	DOH_Y56:=FALSE;
	Y73:=FALSE;	
	//不同蓄能器压力下马大排量电流和主泵供能系数AcPre_w的设置
	IF	GVL_SaveEngine.AI_PAcPre>280 THEN //全部改小0.05
		GVL_SaveEngine.PWM_Y33_SET_Target:=400;//排量120  396-378
		AcPre_w:=0.3;//0.35-0.3 
	ELSIF GVL_SaveEngine.AI_PAcPre>270 THEN
		GVL_SaveEngine.PWM_Y33_SET_Target:=375;//排量130  378-360
		AcPre_w:=0.3;//0.35-0.3//0.15-0.35-0.5-0.4-0.35
	ELSIF GVL_SaveEngine.AI_PAcPre>250 THEN
		GVL_SaveEngine.PWM_Y33_SET_Target:=350;//排量150  340-322 
		AcPre_w:=0.4;//0.4-0.3       //0.25-0.45-0.6-0.5-0.45
	ELSIF  GVL_SaveEngine.AI_PAcPre>230 THEN
		GVL_SaveEngine.PWM_Y33_SET_Target:=325;//排量165 313-295
		AcPre_w:=0.55;//0.5-0.4       //0.4-0.6-0.75-0.65-0.6
	ELSIF  GVL_SaveEngine.AI_PAcPre>220 THEN                               //新增
		GVL_SaveEngine.PWM_Y33_SET_Target:=275;//排量165   
		AcPre_w:=0.6;//0.5-0.4       //0.65
	ELSIF  GVL_SaveEngine.AI_PAcPre>210 THEN
		GVL_SaveEngine.PWM_Y33_SET_Target:=250;//排量190  287-269          //变269-248
		AcPre_w:=0.65;//         //0.55-0.75-0.9-0.8-0.75
	ELSIF GVL_SaveEngine.AI_PAcPre>205 THEN   //200-205 0426
		GVL_SaveEngine.PWM_Y33_SET_Target:=200;//排量200  249-230-248      //248-230
		AcPre_w:=0.7;//         0.6-0.8-0.95-0.85-0.8
	ELSIF GVL_SaveEngine.AI_PAcPre>200 THEN   //190-200 0426
		GVL_SaveEngine.PWM_Y33_SET_Target:=150;//排量210                //230-212
		AcPre_w:=0.75;          //0.7-0.9-1-0.95-0.9
	ELSIF  GVL_SaveEngine.AI_PAcPre>195 THEN  //180-195
		GVL_SaveEngine.PWM_Y33_SET_Target:=100;//排量216                 //230-200
		AcPre_w:=0.85;         //0.85-1
	ELSIF  GVL_SaveEngine.AI_PAcPre>190 THEN  //170-180
		GVL_SaveEngine.PWM_Y33_SET_Target:=100;//排量200
		AcPre_w:=0.9;//0.9-0.8
	ELSIF  GVL_SaveEngine.AI_PAcPre>180 THEN  //160-170
		GVL_SaveEngine.PWM_Y33_SET_Target:=100;//排量200
		AcPre_w:=1;
	ELSE
		GVL_SaveEngine.PWM_Y33_SET_Target:=100;//排量200
		AcPre_w:=1;
	END_IF


	//不同发动机转速下根据马达排量和目标转速计算出的主泵最大电流
  	CASE SPEED_CASE OF
	//                                    权重 速度v 转速n            主卷排量 v_winch
	1: CasePWM_Y1:=REAL_TO_UINT(362.5+47.8*AcPre_w*30/1100*(600-PWM_Y33_SET_Target)/1.85) ;//362.5+1350/转速*AcPre_w*排量
	2: CasePWM_Y1:=REAL_TO_UINT(362.5+47.8*AcPre_w*38/1200*(600-PWM_Y33_SET_Target)/1.85) ;//362.5+1710/转速*AcPre_w*排量
	3: CasePWM_Y1:=REAL_TO_UINT(362.5+47.8*AcPre_w*50/1450*(600-PWM_Y33_SET_Target)/1.85) ;//362.5+2250/转速*AcPre_w*排量
	4: CasePWM_Y1:=REAL_TO_UINT(362.5+47.8*AcPre_w*55/1600*(600-PWM_Y33_SET_Target)/1.85) ;//362.5+2475/转速*AcPre_w*排量
	5: CasePWM_Y1:=REAL_TO_UINT(362.5+47.8*AcPre_w*62/1800*(600-PWM_Y33_SET_Target)/1.85) ;//362.5+2790/转速*AcPre_w*排量
	6: CasePWM_Y1:=REAL_TO_UINT(362.5+47.8*AcPre_w*65/1900*(600-PWM_Y33_SET_Target)/1.85) ;//362.5+2925/转速*AcPre_w*排量
	END_CASE


CasePWM_Y1:=LIMIT(400,CasePWM_Y1,700);
PWM_Y1_Target:=REAL_TO_UINT(UINT_TO_REAL(CasePWM_Y1-PAR_Y1_NegFull)*PWM_JOYY_L_DOWN/1000+PAR_Y1_NegFull);
PWM_Y2_Target:=REAL_TO_UINT(UINT_TO_REAL(CasePWM_Y1-PAR_Y2_NegFull)*PWM_JOYY_L_DOWN/1000+PAR_Y2_NegFull);						

//主阀控制
PWM_Y7_SET_Target:=REAL_TO_UINT(UINT_TO_REAL(PWM_JOYY_L_DOWN)/1000*(PAR_Valve1_PosFull-PAR_Valve2_NegFull)+PAR_Valve2_NegFull);
PWM_Y9_SET_Target:=REAL_TO_UINT(UINT_TO_REAL(PWM_JOYY_L_DOWN)/1000*(PAR_Valve2_PosFull-PAR_Valve2_NegFull)+PAR_Valve2_NegFull);
PWM_Y8_SET:=0;
PWM_Y10_SET:=0;
	
IF PWM_Y33_SET>=PWM_Y33_SET_Target THEN
	PWM_Y33_SET := PWM_Y33_SET_Target;
END_IF
	
IF(PWM_Y33_SET<PWM_Y33_SET_Target) THEN
	PWM_Y33_SET:=REAL_TO_UINT(UINT_TO_REAL(PWM_Y33_SET)+JianGE6);
END_IF

IF DIL_SQ3 THEN
	PWM_Y33_SET:=0;
END_IF
(*主泵功率控制,屏蔽了Pressure_Coe,2模式没有进行恒功率控制，仅保留斜坡*)

//区分发动机转速
MainPump_Pressure_Taget1450:=PAR_NegFull_x;
MainPump_Pressure_Taget1600:=PAR_PosFull_x;
MainPump_Pressure_Taget1750:=PAR_Zero_x;
IF EngineSpeedTarget<=1080 THEN SPEED_CASE:=1;
ELSIF EngineSpeedTarget>1080 AND EngineSpeedTarget<=1300 THEN SPEED_CASE:=2;
ELSIF EngineSpeedTarget>1300 AND EngineSpeedTarget<=1520 THEN SPEED_CASE:=3;
ELSIF EngineSpeedTarget>1520 AND EngineSpeedTarget<=1680 THEN SPEED_CASE:=4;
ELSIF EngineSpeedTarget>1680 AND EngineSpeedTarget<=1820 THEN SPEED_CASE:=5;
ELSIF EngineSpeedTarget>1820 THEN SPEED_CASE:=6;;END_IF
//不同转速下的发动机最大功率*)
CASE SPEED_CASE OF
1:  Enginer_Power:=135;
2:  Enginer_Power:=174;
3:  Enginer_Power:=200;
4:  Enginer_Power:=230;
5:  Enginer_Power:=250;
6:  Enginer_Power:=261;
END_CASE
//不同转速下的压力值
IF(CANO_Fubeng_Press>100)THEN
	CASE SPEED_CASE OF
	1:MainPump_Pressure_Taget:=MainPump_Pressure_Taget1000-HELIU_Press_Target1000;
	2:MainPump_Pressure_Taget:=MainPump_Pressure_Taget1200-HELIU_Press_Target1200;
	3:MainPump_Pressure_Taget:=MainPump_Pressure_Taget1450-HELIU_Press_Target1400;
	4:MainPump_Pressure_Taget:=MainPump_Pressure_Taget1600-HELIU_Press_Target1600;
	5:MainPump_Pressure_Taget:=MainPump_Pressure_Taget1750-HELIU_Press_Target1800;
	6:MainPump_Pressure_Taget:=MainPump_Pressure_Taget1900-HELIU_Press_Target1900;
	END_CASE
ELSE
	CASE SPEED_CASE OF
	1:MainPump_Pressure_Taget:=MainPump_Pressure_Taget1000;
	2:MainPump_Pressure_Taget:=MainPump_Pressure_Taget1200;
	3:MainPump_Pressure_Taget:=MainPump_Pressure_Taget1450;
	4:MainPump_Pressure_Taget:=MainPump_Pressure_Taget1600;
	5:MainPump_Pressure_Taget:=MainPump_Pressure_Taget1750;
	6:MainPump_Pressure_Taget:=MainPump_Pressure_Taget1900;
	END_CASE		
END_IF

IF( CANI_ECOSwitch) THEN
	CASE SPEED_CASE OF
	1:MainPump_Pressure_Taget:=MainPump_Pressure_Taget1000-ECO_Press_Target1000;
	2:MainPump_Pressure_Taget:=MainPump_Pressure_Taget1200-ECO_Press_Target1200;
	3:MainPump_Pressure_Taget:=MainPump_Pressure_Taget1450-ECO_Press_Target1400;
	4:MainPump_Pressure_Taget:=MainPump_Pressure_Taget1600-ECO_Press_Target1600;
	5:MainPump_Pressure_Taget:=MainPump_Pressure_Taget1750-ECO_Press_Target1800;
	6:MainPump_Pressure_Taget:=MainPump_Pressure_Taget1900-ECO_Press_Target1900;
	END_CASE
END_IF
MainPump_Pressure:=CANO_MainPUMP_Press1+CANO_MainPUMP_Press2;
//消除滤波
MainPump_Pressure_Subtract:= UINT_TO_INT(MainPump_Pressure-MainPump_Pressure_last1);


//大范围波动
IF MainPump_Pressure_Subtract>270 OR MainPump_Pressure_Subtract<-270 THEN
	Subtract:=TRUE;
ELSE
	Subtract:=FALSE;	
END_IF
	TIME_LvBo4(IN:=Subtract,PT:=T#10MS);
	
IF(TIME_LvBo4.Q) AND (CANO_MainPUMP_Press1>210) THEN 
		MainPump_Pressure_ChangeBool1:=TRUE;
END_IF
	TIME_LvBo1(IN:=MainPump_Pressure_ChangeBool1,PT:=T#2S);
IF(TIME_LvBo1.Q) THEN
	MainPump_Pressure_ChangeBool1 :=FALSE;
END_IF

IF(MainPump_Pressure_ChangeBool1) AND (MainPump_Pressure>MainPump_Pressure_last1) THEN 
	MainPump_Pressure_last1:=MainPump_Pressure;
END_IF

//小范围波动
t_powertime:=TO_TIME(PAR_DeadBand_x);
IF (NOT MainPump_Pressure_ChangeBool1) THEN
	IF(MainPump_Pressure_Subtract>40 OR MainPump_Pressure_Subtract<-40)THEN 
		MainPump_Pressure_ChangeBool:=TRUE;
	ELSE
		MainPump_Pressure_ChangeBool:=FALSE;
	END_IF

	TIME_LvBo2(IN:=MainPump_Pressure_ChangeBool,PT:=t_powertime);
	IF(TIME_LvBo2.Q )THEN
		MainPump_Pressure_last1:=MainPump_Pressure;
	END_IF	
END_IF


IF PowerHead_move AND NOT(MainWinch_move) THEN
		JianGE2:=0.005;
ELSE
	IF(EngineSpeedTarget>1000 AND EngineSpeedTarget<1300)THEN
		JianGE2:=0.005;
	ELSE
		JianGE2:=0.005;
	END_IF
END_IF
(*	
IF MainPump_Pressure_last1>MainPump_Pressure_Taget THEN
	Pressure_Coe_Taget:=UINT_TO_REAL(MainPump_Pressure_Taget)/UINT_TO_REAL(MainPump_Pressure_last1);(*压力系数*)
ELSE
	Pressure_Coe_Taget:=1;
END_IF
Pressure_Coe := Pressure_Coe_Taget;
*)

(*
Pressure_Coe := 1;
IF MainPump_Pressure_last1>MainPump_Pressure_Taget  THEN
	IF(PWM_Y1_Target>=PAR_Y1_1_NegFull)THEN
		PWM_Y1_Target_OutPut:=REAL_TO_UINT(UINT_TO_REAL(PWM_Y1_Target-PAR_Y1_1_NegFull)*Pressure_Coe+PAR_Y1_1_NegFull);
	END_IF
	IF(PWM_Y2_Target>=PAR_Y1_1_NegFull)THEN
		PWM_Y2_Target_OutPut:=REAL_TO_UINT(UINT_TO_REAL(PWM_Y2_Target-PAR_Y1_1_NegFull)*Pressure_Coe+PAR_Y1_1_NegFull);
	END_IF
ELSE
	PWM_Y1_Target_OutPut:=PWM_Y1_Target;
	PWM_Y2_Target_OutPut:=PWM_Y2_Target;
END_IF
*)

PWM_Y1_Target_OutPut:=PWM_Y1_Target;
PWM_Y2_Target_OutPut:=PWM_Y2_Target;
IF(EngineSpeedTarget>CANO_SPEED AND CANO_SPEED>400)THEN
	EngineSpeedSub:=EngineSpeedTarget - CANO_SPEED;
ELSE
	EngineSpeedSub:=0;
END_IF

IF(PWM_Y1_Target_OutPut<300)THEN PWM_Y1_Target_OutPut:=300;END_IF	
IF(PWM_Y2_Target_OutPut<300)THEN PWM_Y2_Target_OutPut:=300;END_IF

RAMP15_IN:=PWM_Y1_Target_OutPut;
RAMP16_IN:=PWM_Y2_Target_OutPut;
(*
IF MainWinch_move  OR  LeftMove_move OR RightMove_move THEN  
	TIMEBASE_pump:=T#1000MS;
	TIMEBASE_xiehe:=T#500MS;
ELSE
	TIMEBASE_pump:=T#400MS;
	TIMEBASE_xiehe:=T#200MS;
END_IF
t_PowerHead_move(IN:= MainWinch_move,PT:=T#2S);
IF t_PowerHead_move.Q THEN
	F_RAMP_pump:=x_t_PowerHead_move;
	R_RAMP_pump:=x2_t_PowerHead_move;
ELSE
	F_RAMP_pump:=1000;
	R_RAMP_pump:=300;
END_IF
*)
(*
//减斜坡800->2000
RAMP15(
	IN:=UINT_TO_INT(RAMP15_IN), 
	ASCEND:= 300, 
	DESCEND:= 2000, 
	TIMEBASE:=T#1000MS , 
	RESET:=FALSE , 
	OUT=>(PWM_Y1_SET));
	
RAMP16(
	IN:=UINT_TO_INT(RAMP16_IN), 
	ASCEND:= 300, 
	DESCEND:= 2000, 
	TIMEBASE:=T#1000MS , 
	RESET:=FALSE , 
	OUT=>(PWM_Y2_SET));
*)
	CASE SPEED_CASE OF
                1:F_RAMP_pump:=1500; R_RAMP_pump:=100;                  
                2: 		IF MainWinch_move AND (JiaYa_move OR CANO_JiayaPressure>80)  THEN    //3泵同时起压时，降低主泵的加载速度，避免掉速熄火
                                F_RAMP_pump:=1500; R_RAMP_pump:=100;
                        ELSE
                                F_RAMP_pump:=1500; R_RAMP_pump:=100;//从200降
                                IF  PWM_JOYY_L_UP>10 THEN
                                 F_RAMP_pump:=1500; R_RAMP_pump:=200;
                                END_IF
                        END_IF            
                3:
                        IF MainWinch_move AND (JiaYa_move OR CANO_JiayaPressure>80)  THEN    //3泵同时起压时，降低主泵的加载速度，避免掉速熄火
                                F_RAMP_pump:=1500; R_RAMP_pump:=150;
                        ELSE
                                F_RAMP_pump:=1500; R_RAMP_pump:=TO_INT(PAR_NegFull_y);
                                IF  PWM_JOYY_L_UP>10 THEN
                                 F_RAMP_pump:=1500; R_RAMP_pump:=300;
                                END_IF
                        END_IF                
                4:
                        IF MainWinch_move AND (JiaYa_move OR CANO_JiayaPressure>80)  THEN
                                F_RAMP_pump:=1500; R_RAMP_pump:=150;
                        ELSE
                                F_RAMP_pump:=1500; R_RAMP_pump:=TO_INT(PAR_PosFull_y);//从200降
                                IF  PWM_JOYY_L_UP>10 THEN
                                 F_RAMP_pump:=1500; R_RAMP_pump:=300;
                                END_IF
                        END_IF                                
                5:
                        IF MainWinch_move AND (JiaYa_move OR CANO_JiayaPressure>80)  THEN
                                F_RAMP_pump:=1500; R_RAMP_pump:=200;
                        ELSE
                                F_RAMP_pump:=1500; R_RAMP_pump:=TO_INT(PAR_Zero_y);
                                IF  PWM_JOYY_L_UP>10 THEN
                                 F_RAMP_pump:=1500; R_RAMP_pump:=300;
                                END_IF
                        END_IF                        
                6:		IF MainWinch_move AND (JiaYa_move OR CANO_JiayaPressure>80)  THEN
                                F_RAMP_pump:=1500; R_RAMP_pump:=200;
                        ELSE
                                F_RAMP_pump:=1500; R_RAMP_pump:=200;
                                IF  PWM_JOYY_L_UP>10 THEN
                                 F_RAMP_pump:=1500; R_RAMP_pump:=300;
                                END_IF
                        END_IF	
	END_CASE
(******斜坡增步长300 斜坡降步长300->400*****)	
RAMP15(
	IN:=UINT_TO_INT(RAMP15_IN), 
	ASCEND:= R_RAMP_pump, 
	DESCEND:= 2000, //3切2模式时 速度变快 降低主泵电流变化速度 
	TIMEBASE:=T#1000MS , 
	RESET:=FALSE , 
	OUT=>(PWM_Y1_SET));
(******减斜坡300->400*****)	
RAMP16(
	IN:=UINT_TO_INT(RAMP16_IN), 
	ASCEND:= R_RAMP_pump, 
	DESCEND:= 2000, 
	TIMEBASE:=T#1000MS , 
	RESET:=FALSE , 
	OUT=>(PWM_Y2_SET));


IF (NOT Rotation_move) AND (NOT MainWinch_move) AND (NOT PowerHead_move)
		AND (NOT JiaYa_move) AND (NOT ViceWinch_move)
		AND (NOT LeftMove_move) AND (NOT RightMove_move)  THEN
	PWM_Y1_Target:=0;
	PWM_Y2_Target:=0;
END_IF


IF PWM_Y1_SET<TO_INT(PAR_Y1_1_NegFull )THEN
	PWM_Y1_SET:=TO_INT(PAR_Y1_1_NegFull);
END_IF

IF PWM_Y2_SET<TO_INT(PAR_Y1_1_NegFull )THEN
	PWM_Y2_SET:=TO_INT(PAR_Y1_1_NegFull);
END_IF

IF(PWM_Y1_SET>1000) THEN
	PWM_Y1_SET := 300;
END_IF

IF(PWM_Y2_SET>1000) THEN
	PWM_Y2_SET := 300;
END_IF	
  //Y7 8 9 10处理	
		IF(PWM_Y8_SET<1000  AND  PWM_Y8_SET>=900)THEN    //主卷下放斜坡值
				F_RAMP_mainwinch_down:=200;
			
			ELSIF(PWM_Y8_SET<900)THEN
				F_RAMP_mainwinch_down:=400;
			ELSE
				F_RAMP_mainwinch_down:=400;
			END_IF
			
		IF(PWM_Y7_SET<1000  AND  PWM_Y7_SET>=900)THEN  //主卷上提斜坡值
				F_RAMP_mainwinch_down:=300;
		ELSIF(PWM_Y7_SET<900  )THEN
				F_RAMP_mainwinch_down:=200;
		ELSE
				F_RAMP_mainwinch_down:=400;
		END_IF
			
	RAMP7(
		IN:=WORD_TO_INT(PWM_Y7_SET_Target), 
		ASCEND:= R_RAMP_mainwinch, 
		DESCEND:= F_RAMP_mainwinch_up, 
		TIMEBASE:=TIMEBASE_mainwinch , 
		RESET:=FALSE , 
		OUT=>(PWM_Y7_SET_Target1));
	IF(PWM_Y7_SET_Target1>=400) THEN
		Curve_input:=TO_UINT(PWM_Y7_SET_Target1 - 400);
		IF(Curve_input>900) THEN
			Curve_input:=900;
		END_IF
		curve7(input:=REAL_TO_UINT(UINT_TO_REAL(Curve_input)*72.8),Zero:=FALSE,Full:=FALSE,
			   PAR_Progression:=Curve_Par,OutputEnable:=TRUE);
		PWM_Y7_SET:=PAR_Valve1_NegFull + REAL_TO_UINT(UINT_TO_REAL(curve7.Output)/72.8);
	ELSE
		PWM_Y7_SET:=0;
	END_IF
	
(*	
	RAMP8(
		IN:=WORD_TO_INT(PWM_Y8_SET_Target), 
		ASCEND:= R_RAMP_mainwinch, 
		DESCEND:= F_RAMP_mainwinch_down, 
		TIMEBASE:=TIMEBASE_mainwinch , 
		RESET:=FALSE , 
		OUT=>(PWM_Y8_SET_Target1));
	IF(PWM_Y8_SET_Target1>=400) THEN
		Curve_input:=TO_UINT(PWM_Y8_SET_Target1 - 400);
		IF(Curve_input>900) THEN
			Curve_input:=900;
		END_IF
		curve8(input:=REAL_TO_UINT(UINT_TO_REAL(Curve_input)*72.8),Zero:=FALSE,Full:=FALSE,
			   PAR_Progression:=Curve_Par,OutputEnable:=TRUE);
		PWM_Y8_SET:=PAR_Valve1_NegFull + REAL_TO_UINT(UINT_TO_REAL(curve8.Output)/72.8);
	ELSE
		PWM_Y8_SET:=0;
	END_IF
*)	
	
	RAMP9(
		IN:=WORD_TO_INT(PWM_Y9_SET_Target), 
		ASCEND:= R_RAMP_mainwinch, 
		DESCEND:= F_RAMP_mainwinch_up, 
		TIMEBASE:=TIMEBASE_mainwinch , 
		RESET:=FALSE , 
		OUT=>(PWM_Y9_SET_Target1));
	IF(PWM_Y9_SET_Target1>=400) THEN
		Curve_input:=TO_UINT(PWM_Y9_SET_Target1 - 400);
		IF(Curve_input>900) THEN
			Curve_input:=900;
		END_IF
		curve9(input:=REAL_TO_UINT(UINT_TO_REAL(Curve_input)*72.8),Zero:=FALSE,Full:=FALSE,
			   PAR_Progression:=Curve_Par,OutputEnable:=TRUE);
		PWM_Y9_SET:=PAR_Valve1_NegFull + REAL_TO_UINT(UINT_TO_REAL(curve9.Output)/72.8);
	ELSE
		PWM_Y9_SET:=0;
	END_IF
(*	
	RAMP10(
		IN:=WORD_TO_INT(PWM_Y10_SET_Target), 
		ASCEND:= R_RAMP_mainwinch, 
		DESCEND:= F_RAMP_mainwinch_down, 
		TIMEBASE:=TIMEBASE_mainwinch , 
		RESET:=FALSE , 
		OUT=>(PWM_Y10_SET_Target1));
	IF(PWM_Y10_SET_Target1>=400) THEN
		Curve_input:=TO_UINT(PWM_Y10_SET_Target1 - 400);
		IF(Curve_input>900) THEN
			Curve_input:=900;
		END_IF
		curve10(input:=REAL_TO_UINT(UINT_TO_REAL(Curve_input)*72.8),Zero:=FALSE,Full:=FALSE,
			   PAR_Progression:=Curve_Par,OutputEnable:=TRUE);
		PWM_Y10_SET:=PAR_Valve1_NegFull + REAL_TO_UINT(UINT_TO_REAL(curve10.Output)/72.8);
	ELSE
		PWM_Y10_SET:=0;
	END_IF
*)
    //Y7 8 9 10范围限制
	IF(PWM_Y7_SET>1300)THEN
		PWM_Y7_SET :=1300;
	END_IF
	IF(PWM_Y8_SET>1300)THEN
		PWM_Y8_SET :=1300;
	END_IF
	IF(PWM_Y9_SET>1300)THEN
		PWM_Y9_SET :=1300;
	END_IF
	IF(PWM_Y10_SET>1300)THEN
		PWM_Y10_SET :=1300;
	END_IF
	
	IF(PWM_Y7_SET<=300)THEN
		PWM_Y7_SET :=0;
	END_IF
	IF(PWM_Y8_SET<=300)THEN
		PWM_Y8_SET :=0;
	END_IF
	IF(PWM_Y9_SET<=300)THEN
		PWM_Y9_SET :=0;
	END_IF
	IF(PWM_Y10_SET<=300)THEN
		PWM_Y10_SET :=0;
	END_IF
	(*主泵卸荷阀控制*)
		//PWM_Y39_SET_Target:=MAX(PWM_Y8_SET,PWM_Y7_SET_Target);//直接给输出卸荷
		PWM_Y40_SET_Target:=MAX(PWM_Y9_SET_Target,PWM_Y10_SET);
	//(*卸荷动作缓冲*)
(*RAMP19(
	IN:=WORD_TO_INT(PWM_Y39_SET_Target), 
	ASCEND:= R_RAMP_xiehe, 
	DESCEND:= F_RAMP_xiehe, 
	TIMEBASE:=TIMEBASE_xiehe , 
	RESET:=FALSE , 
	OUT=>(PWM_Y39_SET_Target1));
IF(PWM_Y39_SET_Target1>=400) THEN
	Curve_input:=TO_UINT(PWM_Y39_SET_Target1 - 400);
	IF(Curve_input>900) THEN
		Curve_input:=900;
	END_IF
	curve19(input:=REAL_TO_UINT(UINT_TO_REAL(Curve_input)*72.8),Zero:=FALSE,Full:=FALSE,
		   PAR_Progression:=Curve_Par1,OutputEnable:=TRUE);
	PWM_Y39_SET:=PAR_Valve1_NegFull + REAL_TO_UINT(UINT_TO_REAL(curve19.Output)/72.8);
ELSE
	PWM_Y39_SET:=0;
END_IF
*)

RAMP20(
	IN:=WORD_TO_INT(PWM_Y40_SET_Target), 
	ASCEND:= R_RAMP_xiehe, 
	DESCEND:= F_RAMP_xiehe, 
	TIMEBASE:=TIMEBASE_xiehe , 
	RESET:=FALSE , 
	OUT=>(PWM_Y40_SET_Target1));
IF(PWM_Y40_SET_Target1>=400) THEN
	Curve_input:=TO_UINT(PWM_Y40_SET_Target1 - 400);
	IF(Curve_input>900) THEN
		Curve_input:=900;
	END_IF
	curve20(input:=REAL_TO_UINT(UINT_TO_REAL(Curve_input)*72.8),Zero:=FALSE,Full:=FALSE,
		   PAR_Progression:=Curve_Par1,OutputEnable:=TRUE);
	PWM_Y40_SET:=PAR_Valve1_NegFull + REAL_TO_UINT(UINT_TO_REAL(curve20.Output)/72.8);
ELSE
	PWM_Y40_SET:=0;
END_IF

IF(PWM_Y39_SET>1300)THEN
	PWM_Y39_SET :=1300;
END_IF
IF(PWM_Y40_SET>1300)THEN
	PWM_Y40_SET :=1300;
END_IF

IF(PWM_Y39_SET<=300)THEN
	PWM_Y39_SET :=0;
END_IF
IF(PWM_Y40_SET<=300)THEN
	PWM_Y40_SET :=0;
END_IF

END_PROGRAM

// StandardPLC/Application/SaveEngine/SaveEngineMode_3
PROGRAM SaveEngineMode_3
VAR
	PressLvBo_TON:TON;
	PressLvBo_TON1: TON;
	PressLvBo_TON2: TON;
	PressLvBo_TON3: TON;

END_VAR


(*******************节能控制阀主阀主泵输出执行**************************)
	
//ELSIF(GVL_SaveEngine.SaveEngineMode=3)THEN//上升能量不足模式
	GVL_SaveEngine.Y72OutPutState:=0;
	GVL_SaveEngine.Y71OutPutState:=0;
	DOH_Y56:=FALSE;
		Y73:=FALSE;	
	PWM_Y1_Target:=REAL_TO_UINT(UINT_TO_REAL(PWM_JOYY_L_DOWN)/1000*0.9*(PAR_Y1_PosFull-PAR_Y1_NegFull)+PAR_Y1_NegFull);
	PWM_Y2_Target:=REAL_TO_UINT(UINT_TO_REAL(PWM_JOYY_L_DOWN)/1000*0.9*(PAR_Y2_PosFull-PAR_Y2_NegFull)+PAR_Y2_NegFull);
	PWM_Y7_SET_Target:=REAL_TO_UINT(UINT_TO_REAL(PWM_JOYY_L_DOWN)/1000*(PAR_Valve1_PosFull-PAR_Valve2_NegFull)+PAR_Valve2_NegFull);
	PWM_Y9_SET_Target:=REAL_TO_UINT(UINT_TO_REAL(PWM_JOYY_L_DOWN)/1000*(PAR_Valve2_PosFull-PAR_Valve2_NegFull)+PAR_Valve2_NegFull);
	PWM_Y8_SET_Target:=300;
	PWM_Y10_SET_Target:=300;		
	(*电控马达主卷变量控制*)
	
PressLvBo_TON(IN:=CANO_ZhuJuanPressure>310,PT:=T#300MS);
PressLvBo_TON1(IN:=CANO_ZhuJuanPressure>290 AND CANO_ZhuJuanPressure<=310,PT:=T#300MS);
PressLvBo_TON2(IN:=CANO_ZhuJuanPressure>270 AND CANO_ZhuJuanPressure<=290,PT:=T#300MS);
PressLvBo_TON3(IN:=CANO_ZhuJuanPressure>250 AND CANO_ZhuJuanPressure<=270,PT:=T#300MS);
IF(CANO_ZhuJuanPressure>310 AND PressLvBo_TON.Q) OR P31_Flag THEN
        PWM_Y33_SET_Target :=230;   //排量200
        P31_Flag:=TRUE;
        IF (CANO_ZhuJuanPressure<270) THEN
                P31_Flag:=FALSE;        
        END_IF
ELSIF(CANO_ZhuJuanPressure>290 AND PressLvBo_TON1.Q) OR P29_Flag THEN   
        PWM_Y33_SET_Target :=267;   //排量180
        P29_Flag:=TRUE; 
        IF (CANO_ZhuJuanPressure<250) THEN
                P29_Flag:=FALSE; 
        END_IF
ELSIF(CANO_ZhuJuanPressure>270 AND PressLvBo_TON2.Q) OR P27_Flag THEN   
        PWM_Y33_SET_Target :=304;  //排量160
        P27_Flag:=TRUE;
        IF (CANO_ZhuJuanPressure<230) THEN
                P27_Flag:=FALSE; 
        END_IF
ELSIF(CANO_ZhuJuanPressure>250 AND PressLvBo_TON3.Q) OR P25_Flag THEN //压力小于270   
        PWM_Y33_SET_Target :=340;  //排量140
        P25_Flag:=TRUE; 
        IF (CANO_ZhuJuanPressure<210) THEN
                P25_Flag:=FALSE; 
        END_IF
ELSE //(CANO_ZhuJuanPressure<=250) THEN
        PWM_Y33_SET_Target :=370;
END_IF
	(*IF BiaoZHI_MainWinchUp THEN
		PWM_Y33_SET_Target:=370;
	END_IF
	*)
	  //Y33输出处理
	IF PWM_Y33_SET>=PWM_Y33_SET_Target THEN
	PWM_Y33_SET := PWM_Y33_SET_Target;
	END_IF
		
	IF(PWM_Y33_SET<PWM_Y33_SET_Target) THEN
		PWM_Y33_SET:=REAL_TO_UINT(UINT_TO_REAL(PWM_Y33_SET)+JianGE6);
	END_IF
	
	IF DIL_SQ3 THEN
		PWM_Y33_SET:=0;
	END_IF
	
(*主泵功率控制*)

//区分发动机转速
MainPump_Pressure_Taget1450:=PAR_NegFull_x;
MainPump_Pressure_Taget1600:=PAR_PosFull_x;
MainPump_Pressure_Taget1750:=PAR_Zero_x;
IF EngineSpeedTarget<=1080 THEN SPEED_CASE:=1;
ELSIF EngineSpeedTarget>1080 AND EngineSpeedTarget<=1300 THEN SPEED_CASE:=2;
ELSIF EngineSpeedTarget>1300 AND EngineSpeedTarget<=1520 THEN SPEED_CASE:=3;
ELSIF EngineSpeedTarget>1520 AND EngineSpeedTarget<=1680 THEN SPEED_CASE:=4;
ELSIF EngineSpeedTarget>1680 AND EngineSpeedTarget<=1820 THEN SPEED_CASE:=5;
ELSIF EngineSpeedTarget>1820 THEN SPEED_CASE:=6;;END_IF
//不同转速下的发动机最大功率*)
CASE SPEED_CASE OF
1:  Enginer_Power:=135;
2:  Enginer_Power:=174;
3:  Enginer_Power:=200;
4:  Enginer_Power:=230;
5:  Enginer_Power:=250;
6:  Enginer_Power:=261;
END_CASE
//不同转速下的压力值
IF(CANO_Fubeng_Press>100)THEN
	CASE SPEED_CASE OF
	1:MainPump_Pressure_Taget:=MainPump_Pressure_Taget1000-HELIU_Press_Target1000;
	2:MainPump_Pressure_Taget:=MainPump_Pressure_Taget1200-HELIU_Press_Target1200;
	3:MainPump_Pressure_Taget:=MainPump_Pressure_Taget1450-HELIU_Press_Target1400;
	4:MainPump_Pressure_Taget:=MainPump_Pressure_Taget1600-HELIU_Press_Target1600;
	5:MainPump_Pressure_Taget:=MainPump_Pressure_Taget1750-HELIU_Press_Target1800;
	6:MainPump_Pressure_Taget:=MainPump_Pressure_Taget1900-HELIU_Press_Target1900;
	END_CASE
ELSE
	CASE SPEED_CASE OF
	1:MainPump_Pressure_Taget:=MainPump_Pressure_Taget1000;
	2:MainPump_Pressure_Taget:=MainPump_Pressure_Taget1200;
	3:MainPump_Pressure_Taget:=MainPump_Pressure_Taget1450;
	4:MainPump_Pressure_Taget:=MainPump_Pressure_Taget1600;
	5:MainPump_Pressure_Taget:=MainPump_Pressure_Taget1750;
	6:MainPump_Pressure_Taget:=MainPump_Pressure_Taget1900;
	END_CASE		
END_IF

IF( CANI_ECOSwitch) THEN
	CASE SPEED_CASE OF
	1:MainPump_Pressure_Taget:=MainPump_Pressure_Taget1000-ECO_Press_Target1000;
	2:MainPump_Pressure_Taget:=MainPump_Pressure_Taget1200-ECO_Press_Target1200;
	3:MainPump_Pressure_Taget:=MainPump_Pressure_Taget1450-ECO_Press_Target1400;
	4:MainPump_Pressure_Taget:=MainPump_Pressure_Taget1600-ECO_Press_Target1600;
	5:MainPump_Pressure_Taget:=MainPump_Pressure_Taget1750-ECO_Press_Target1800;
	6:MainPump_Pressure_Taget:=MainPump_Pressure_Taget1900-ECO_Press_Target1900;
	END_CASE
END_IF
MainPump_Pressure:=CANO_MainPUMP_Press1+CANO_MainPUMP_Press2;
//消除滤波
MainPump_Pressure_Subtract:= UINT_TO_INT(MainPump_Pressure-MainPump_Pressure_last1);


//大范围波动
IF MainPump_Pressure_Subtract>270 OR MainPump_Pressure_Subtract<-270 THEN
	Subtract:=TRUE;
ELSE
	Subtract:=FALSE;	
END_IF
	TIME_LvBo4(IN:=Subtract,PT:=T#10MS);
	
IF(TIME_LvBo4.Q) AND (CANO_MainPUMP_Press1>210) THEN 
	MainPump_Pressure_ChangeBool1:=TRUE;
END_IF
	TIME_LvBo1(IN:=MainPump_Pressure_ChangeBool1,PT:=T#2S);
IF(TIME_LvBo1.Q) THEN
	MainPump_Pressure_ChangeBool1 :=FALSE;
END_IF

IF(MainPump_Pressure_ChangeBool1) AND (MainPump_Pressure>MainPump_Pressure_last1) THEN 
	MainPump_Pressure_last1:=MainPump_Pressure;
END_IF

//小范围波动
t_powertime:=TO_TIME(PAR_DeadBand_x);
IF (NOT MainPump_Pressure_ChangeBool1) THEN
	IF(MainPump_Pressure_Subtract>40 OR MainPump_Pressure_Subtract<-40)THEN 
		MainPump_Pressure_ChangeBool:=TRUE;
	ELSE
		MainPump_Pressure_ChangeBool:=FALSE;
	END_IF

	TIME_LvBo2(IN:=MainPump_Pressure_ChangeBool,PT:=t_powertime);
	IF(TIME_LvBo2.Q )THEN
		MainPump_Pressure_last1:=MainPump_Pressure;
	END_IF	
END_IF


IF PowerHead_move AND NOT(MainWinch_move) THEN
		JianGE2:=0.005;
ELSE
	IF(EngineSpeedTarget>1000 AND EngineSpeedTarget<1300)THEN
		JianGE2:=0.005;
	ELSE
		JianGE2:=0.005;
	END_IF
END_IF

IF MainPump_Pressure_last1>MainPump_Pressure_Taget THEN
	Pressure_Coe_Taget:=UINT_TO_REAL(MainPump_Pressure_Taget)/UINT_TO_REAL(MainPump_Pressure_last1);(*压力系数*)
ELSE
	Pressure_Coe_Taget:=1;
END_IF
Pressure_Coe := Pressure_Coe_Taget;


IF MainPump_Pressure_last1>MainPump_Pressure_Taget  THEN
	IF(PWM_Y1_Target>=PAR_Y1_1_NegFull)THEN
		PWM_Y1_Target_OutPut:=REAL_TO_UINT(UINT_TO_REAL(PWM_Y1_Target-PAR_Y1_1_NegFull)*Pressure_Coe+PAR_Y1_1_NegFull);
	END_IF
	IF(PWM_Y2_Target>=PAR_Y1_1_NegFull)THEN
		PWM_Y2_Target_OutPut:=REAL_TO_UINT(UINT_TO_REAL(PWM_Y2_Target-PAR_Y1_1_NegFull)*Pressure_Coe+PAR_Y1_1_NegFull);
	END_IF
ELSE
	PWM_Y1_Target_OutPut:=PWM_Y1_Target;
	PWM_Y2_Target_OutPut:=PWM_Y2_Target;
END_IF
//PWM_Y1_Target_OutPut:=PWM_Y1_Target;
//PWM_Y2_Target_OutPut:=PWM_Y2_Target;


IF(EngineSpeedTarget>CANO_SPEED AND CANO_SPEED>400)THEN
	EngineSpeedSub:=EngineSpeedTarget - CANO_SPEED;
ELSE
	EngineSpeedSub:=0;
END_IF

IF(PWM_Y1_Target_OutPut<300)THEN PWM_Y1_Target_OutPut:=300;END_IF	
IF(PWM_Y2_Target_OutPut<300)THEN PWM_Y2_Target_OutPut:=300;END_IF

RAMP15_IN:=PWM_Y1_Target_OutPut;
RAMP16_IN:=PWM_Y2_Target_OutPut;
(*
IF MainWinch_move  OR  LeftMove_move OR RightMove_move THEN  
	TIMEBASE_pump:=T#1000MS;
	TIMEBASE_xiehe:=T#500MS;
ELSE
	TIMEBASE_pump:=T#400MS;
	TIMEBASE_xiehe:=T#200MS;
END_IF
t_PowerHead_move(IN:= MainWinch_move,PT:=T#2S);
IF t_PowerHead_move.Q THEN
	F_RAMP_pump:=x_t_PowerHead_move;
	R_RAMP_pump:=x2_t_PowerHead_move;
ELSE
	F_RAMP_pump:=1000;
	R_RAMP_pump:=300;
END_IF
*)

(*
RAMP15(
	IN:=UINT_TO_INT(RAMP15_IN), 
	ASCEND:= 300, 
	DESCEND:= 400, 
	TIMEBASE:=T#1000MS , 
	RESET:=FALSE , 
	OUT=>(PWM_Y1_SET));
	
RAMP16(
	IN:=UINT_TO_INT(RAMP16_IN), 
	ASCEND:= 300, 
	DESCEND:= 400, 
	TIMEBASE:=T#1000MS , 
	RESET:=FALSE , 
	OUT=>(PWM_Y2_SET));
*)
	CASE SPEED_CASE OF
                1:F_RAMP_pump:=1500; R_RAMP_pump:=100;                  
                2: 		IF MainWinch_move AND (JiaYa_move OR CANO_JiayaPressure>80)  THEN    //3泵同时起压时，降低主泵的加载速度，避免掉速熄火
                                F_RAMP_pump:=1500; R_RAMP_pump:=100;
                        ELSE
                                F_RAMP_pump:=1500; R_RAMP_pump:=100;//从200降
                                IF  PWM_JOYY_L_UP>10 THEN
                                 F_RAMP_pump:=1500; R_RAMP_pump:=200;
                                END_IF
                        END_IF            
                3:
                        IF MainWinch_move AND (JiaYa_move OR CANO_JiayaPressure>80)  THEN    //3泵同时起压时，降低主泵的加载速度，避免掉速熄火
                                F_RAMP_pump:=1500; R_RAMP_pump:=150;
                        ELSE
                                F_RAMP_pump:=1500; R_RAMP_pump:=TO_INT(PAR_NegFull_y);
                                IF  PWM_JOYY_L_UP>10 THEN
                                 F_RAMP_pump:=1500; R_RAMP_pump:=300;
                                END_IF
                        END_IF                
                4:
                        IF MainWinch_move AND (JiaYa_move OR CANO_JiayaPressure>80)  THEN
                                F_RAMP_pump:=1500; R_RAMP_pump:=150;
                        ELSE
                                F_RAMP_pump:=1500; R_RAMP_pump:=TO_INT(PAR_PosFull_y);//从200降
                                IF  PWM_JOYY_L_UP>10 THEN
                                 F_RAMP_pump:=1500; R_RAMP_pump:=300;
                                END_IF
                        END_IF                                
                5:
                        IF MainWinch_move AND (JiaYa_move OR CANO_JiayaPressure>80)  THEN
                                F_RAMP_pump:=1500; R_RAMP_pump:=200;
                        ELSE
                                F_RAMP_pump:=1500; R_RAMP_pump:=TO_INT(PAR_Zero_y);
                                IF  PWM_JOYY_L_UP>10 THEN
                                 F_RAMP_pump:=1500; R_RAMP_pump:=300;
                                END_IF
                        END_IF                        
                6:		IF MainWinch_move AND (JiaYa_move OR CANO_JiayaPressure>80)  THEN
                                F_RAMP_pump:=1500; R_RAMP_pump:=200;
                        ELSE
                                F_RAMP_pump:=1500; R_RAMP_pump:=200;
                                IF  PWM_JOYY_L_UP>10 THEN
                                 F_RAMP_pump:=1500; R_RAMP_pump:=300;
                                END_IF
                        END_IF
	END_CASE
(******斜坡增步长300 斜坡降步长300->400*****)	
RAMP15(
	IN:=UINT_TO_INT(RAMP15_IN), 
	ASCEND:= R_RAMP_pump, 
	DESCEND:= 1500, 
	TIMEBASE:=T#1000MS , 
	RESET:=FALSE , 
	OUT=>(PWM_Y1_SET));
(******减斜坡300->400*****)	
RAMP16(
	IN:=UINT_TO_INT(RAMP16_IN), 
	ASCEND:= R_RAMP_pump, 
	DESCEND:= 1500, 
	TIMEBASE:=T#1000MS , 
	RESET:=FALSE , 
	OUT=>(PWM_Y2_SET));


IF (NOT Rotation_move) AND (NOT MainWinch_move) AND (NOT PowerHead_move)
		AND (NOT JiaYa_move) AND (NOT ViceWinch_move)
		AND (NOT LeftMove_move) AND (NOT RightMove_move)  THEN
	PWM_Y1_Target:=0;
	PWM_Y2_Target:=0;
END_IF


IF PWM_Y1_SET<TO_INT(PAR_Y1_1_NegFull )THEN
	PWM_Y1_SET:=TO_INT(PAR_Y1_1_NegFull);
END_IF

IF PWM_Y2_SET<TO_INT(PAR_Y1_1_NegFull )THEN
	PWM_Y2_SET:=TO_INT(PAR_Y1_1_NegFull);
END_IF

IF(PWM_Y1_SET>1000) THEN
	PWM_Y1_SET := 300;
END_IF

IF(PWM_Y2_SET>1000) THEN
	PWM_Y2_SET := 300;
END_IF		
  //Y7 8 9 10处理	
		IF(PWM_Y8_SET<1000  AND  PWM_Y8_SET>=900)THEN    //主卷下放斜坡值
				F_RAMP_mainwinch_down:=200;
			
			ELSIF(PWM_Y8_SET<900)THEN
				F_RAMP_mainwinch_down:=400;
			ELSE
				F_RAMP_mainwinch_down:=400;
			END_IF
			
		IF(PWM_Y7_SET<1000  AND  PWM_Y7_SET>=900)THEN  //主卷上提斜坡值
				F_RAMP_mainwinch_down:=300;
		ELSIF(PWM_Y7_SET<900  )THEN
				F_RAMP_mainwinch_down:=200;
		ELSE
				F_RAMP_mainwinch_down:=400;
		END_IF
			
	RAMP7(
		IN:=WORD_TO_INT(PWM_Y7_SET_Target), 
		ASCEND:= R_RAMP_mainwinch, 
		DESCEND:= F_RAMP_mainwinch_up, 
		TIMEBASE:=TIMEBASE_mainwinch , 
		RESET:=FALSE , 
		OUT=>(PWM_Y7_SET_Target1));
	IF(PWM_Y7_SET_Target1>=400) THEN
		Curve_input:=TO_UINT(PWM_Y7_SET_Target1 - 400);
		IF(Curve_input>900) THEN
			Curve_input:=900;
		END_IF
		curve7(input:=REAL_TO_UINT(UINT_TO_REAL(Curve_input)*72.8),Zero:=FALSE,Full:=FALSE,
			   PAR_Progression:=Curve_Par,OutputEnable:=TRUE);
		PWM_Y7_SET:=PAR_Valve1_NegFull + REAL_TO_UINT(UINT_TO_REAL(curve7.Output)/72.8);
	ELSE
		PWM_Y7_SET:=0;
	END_IF
	
		PWM_Y8_SET:=0;
	
	RAMP9(
		IN:=WORD_TO_INT(PWM_Y9_SET_Target), 
		ASCEND:= R_RAMP_mainwinch, 
		DESCEND:= F_RAMP_mainwinch_up, 
		TIMEBASE:=TIMEBASE_mainwinch , 
		RESET:=FALSE , 
		OUT=>(PWM_Y9_SET_Target1));
	IF(PWM_Y9_SET_Target1>=400) THEN
		Curve_input:=TO_UINT(PWM_Y9_SET_Target1 - 400);
		IF(Curve_input>900) THEN
			Curve_input:=900;
		END_IF
		curve9(input:=REAL_TO_UINT(UINT_TO_REAL(Curve_input)*72.8),Zero:=FALSE,Full:=FALSE,
			   PAR_Progression:=Curve_Par,OutputEnable:=TRUE);
		PWM_Y9_SET:=PAR_Valve1_NegFull + REAL_TO_UINT(UINT_TO_REAL(curve9.Output)/72.8);
	ELSE
		PWM_Y9_SET:=0;
	END_IF
	
		PWM_Y10_SET:=0;
    //Y7 8 9 10范围限制
	IF(PWM_Y7_SET>1300)THEN
		PWM_Y7_SET :=1300;
	END_IF
	IF(PWM_Y8_SET>1300)THEN
		PWM_Y8_SET :=1300;
	END_IF
	IF(PWM_Y9_SET>1300)THEN
		PWM_Y9_SET :=1300;
	END_IF
	IF(PWM_Y10_SET>1300)THEN
		PWM_Y10_SET :=1300;
	END_IF
	
	IF(PWM_Y7_SET<=300)THEN
		PWM_Y7_SET :=0;
	END_IF
	IF(PWM_Y8_SET<=300)THEN
		PWM_Y8_SET :=0;
	END_IF
	IF(PWM_Y9_SET<=300)THEN
		PWM_Y9_SET :=0;
	END_IF
	IF(PWM_Y10_SET<=300)THEN
		PWM_Y10_SET :=0;
	END_IF
	(*主泵卸荷阀控制*)
		PWM_Y39_SET_Target:=PWM_Y7_SET_Target;
		PWM_Y40_SET_Target:=PWM_Y9_SET_Target;
	(*卸荷动作缓冲*)
RAMP19(
	IN:=WORD_TO_INT(PWM_Y39_SET_Target), 
	ASCEND:= R_RAMP_xiehe, 
	DESCEND:= F_RAMP_xiehe, 
	TIMEBASE:=TIMEBASE_xiehe , 
	RESET:=FALSE , 
	OUT=>(PWM_Y39_SET_Target1));
IF(PWM_Y39_SET_Target1>=400) THEN
	Curve_input:=TO_UINT(PWM_Y39_SET_Target1 - 400);
	IF(Curve_input>900) THEN
		Curve_input:=900;
	END_IF
	curve19(input:=REAL_TO_UINT(UINT_TO_REAL(Curve_input)*72.8),Zero:=FALSE,Full:=FALSE,
		   PAR_Progression:=Curve_Par1,OutputEnable:=TRUE);
	PWM_Y39_SET:=PAR_Valve1_NegFull + REAL_TO_UINT(UINT_TO_REAL(curve19.Output)/72.8);
ELSE
	PWM_Y39_SET:=0;
END_IF


RAMP20(
	IN:=WORD_TO_INT(PWM_Y40_SET_Target), 
	ASCEND:= R_RAMP_xiehe, 
	DESCEND:= F_RAMP_xiehe, 
	TIMEBASE:=TIMEBASE_xiehe , 
	RESET:=FALSE , 
	OUT=>(PWM_Y40_SET_Target1));
IF(PWM_Y40_SET_Target1>=400) THEN
	Curve_input:=TO_UINT(PWM_Y40_SET_Target1 - 400);
	IF(Curve_input>900) THEN
		Curve_input:=900;
	END_IF
	curve20(input:=REAL_TO_UINT(UINT_TO_REAL(Curve_input)*72.8),Zero:=FALSE,Full:=FALSE,
		   PAR_Progression:=Curve_Par1,OutputEnable:=TRUE);
	PWM_Y40_SET:=PAR_Valve1_NegFull + REAL_TO_UINT(UINT_TO_REAL(curve20.Output)/72.8);
ELSE
	PWM_Y40_SET:=0;
END_IF
	
IF(PWM_Y39_SET>1300)THEN
	PWM_Y39_SET :=1300;
END_IF
IF(PWM_Y40_SET>1300)THEN
	PWM_Y40_SET :=1300;
END_IF

IF(PWM_Y39_SET<=300)THEN
	PWM_Y39_SET :=0;
END_IF
IF(PWM_Y40_SET<=300)THEN
	PWM_Y40_SET :=0;
END_IF

END_PROGRAM

// StandardPLC/Application/SaveEngine/SaveEngineMode_4
PROGRAM SaveEngineMode_4
VAR

END_VAR


(*******************节能控制阀主阀主泵输出执行**************************)
//ELSIF(GVL_SaveEngine.SaveEngineMode=4)THEN//中位模式
	GVL_SaveEngine.Y72OutPutState:=0;
	GVL_SaveEngine.Y71OutPutState:=0;	
	DOH_Y56:=FALSE;
	Y73:=FALSE;	
	//PWM_Y8_SET:=0;
	//PWM_Y10_SET:=0;
	//PWM_Y8_SET_Target:=0;
	//PWM_Y10_SET_Target:=0;
	//增加下降斜坡  防止M1下降回中位的时候过高
	PWM_Y7_SET_Target:=0;
	PWM_Y9_SET_Target:=0;
	PWM_Y8_SET_Target:=0;
	PWM_Y10_SET_Target:=0;
	RAMP7(
		IN:=WORD_TO_INT(PWM_Y7_SET_Target), 
		ASCEND:= R_RAMP_mainwinch, 
		DESCEND:= F_RAMP_mainwinch_up, 
		TIMEBASE:=TIMEBASE_mainwinch , 
		RESET:=FALSE , 
		OUT=>(PWM_Y7_SET_Target1));
	IF(PWM_Y7_SET_Target1>=400) THEN
		Curve_input:=TO_UINT(PWM_Y7_SET_Target1 - 400);
		IF(Curve_input>900) THEN
			Curve_input:=900;
		END_IF
		curve7(input:=REAL_TO_UINT(UINT_TO_REAL(Curve_input)*72.8),Zero:=FALSE,Full:=FALSE,
			   PAR_Progression:=Curve_Par,OutputEnable:=TRUE);
		PWM_Y7_SET:=PAR_Valve1_NegFull + REAL_TO_UINT(UINT_TO_REAL(curve7.Output)/72.8);
	ELSE
		PWM_Y7_SET:=0;
	END_IF
	
	RAMP8(
		IN:=WORD_TO_INT(PWM_Y8_SET_Target), 
		ASCEND:= R_RAMP_mainwinch, 
		DESCEND:= F_RAMP_mainwinch_down, 
		TIMEBASE:=TIMEBASE_mainwinch , 
		RESET:=FALSE , 
		OUT=>(PWM_Y8_SET_Target1));
	IF(PWM_Y8_SET_Target1>=400) THEN
		Curve_input:=TO_UINT(PWM_Y8_SET_Target1 - 400);
		IF(Curve_input>900) THEN
			Curve_input:=900;
		END_IF
		curve8(input:=REAL_TO_UINT(UINT_TO_REAL(Curve_input)*72.8),Zero:=FALSE,Full:=FALSE,
			   PAR_Progression:=Curve_Par,OutputEnable:=TRUE);
		PWM_Y8_SET:=PAR_Valve1_NegFull + REAL_TO_UINT(UINT_TO_REAL(curve8.Output)/72.8);
	ELSE
		PWM_Y8_SET:=0;
	END_IF
		RAMP9(
		IN:=WORD_TO_INT(PWM_Y9_SET_Target), 
		ASCEND:= R_RAMP_mainwinch, 
		DESCEND:= F_RAMP_mainwinch_up, 
		TIMEBASE:=TIMEBASE_mainwinch , 
		RESET:=FALSE , 
		OUT=>(PWM_Y9_SET_Target1));
	IF(PWM_Y9_SET_Target1>=400) THEN
		Curve_input:=TO_UINT(PWM_Y9_SET_Target1 - 400);
		IF(Curve_input>900) THEN
			Curve_input:=900;
		END_IF
		curve9(input:=REAL_TO_UINT(UINT_TO_REAL(Curve_input)*72.8),Zero:=FALSE,Full:=FALSE,
			   PAR_Progression:=Curve_Par,OutputEnable:=TRUE);
		PWM_Y9_SET:=PAR_Valve1_NegFull + REAL_TO_UINT(UINT_TO_REAL(curve9.Output)/72.8);
	ELSE
		PWM_Y9_SET:=0;
	END_IF
	
	RAMP10(
		IN:=WORD_TO_INT(PWM_Y10_SET_Target), 
		ASCEND:= R_RAMP_mainwinch, 
		DESCEND:= F_RAMP_mainwinch_down, 
		TIMEBASE:=TIMEBASE_mainwinch , 
		RESET:=FALSE , 
		OUT=>(PWM_Y10_SET_Target1));
	IF(PWM_Y10_SET_Target1>=400) THEN
		Curve_input:=TO_UINT(PWM_Y10_SET_Target1 - 400);
		IF(Curve_input>900) THEN
			Curve_input:=900;
		END_IF
		curve10(input:=REAL_TO_UINT(UINT_TO_REAL(Curve_input)*72.8),Zero:=FALSE,Full:=FALSE,
			   PAR_Progression:=Curve_Par,OutputEnable:=TRUE);
		PWM_Y10_SET:=PAR_Valve1_NegFull + REAL_TO_UINT(UINT_TO_REAL(curve10.Output)/72.8);
	ELSE
		PWM_Y10_SET:=0;
	END_IF
    //Y7 8 9 10范围限制
	IF(PWM_Y7_SET>1300)THEN
		PWM_Y7_SET :=1300;
	END_IF
	IF(PWM_Y8_SET>1300)THEN
		PWM_Y8_SET :=1300;
	END_IF
	IF(PWM_Y9_SET>1300)THEN
		PWM_Y9_SET :=1300;
	END_IF
	IF(PWM_Y10_SET>1300)THEN
		PWM_Y10_SET :=1300;
	END_IF
	
	IF(PWM_Y7_SET<=300)THEN
		PWM_Y7_SET :=0;
	END_IF
	IF(PWM_Y8_SET<=300)THEN
		PWM_Y8_SET :=0;
	END_IF
	IF(PWM_Y9_SET<=300)THEN
		PWM_Y9_SET :=0;
	END_IF
	IF(PWM_Y10_SET<=300)THEN
		PWM_Y10_SET :=0;
	END_IF

	
	
	//PWM_Y7_SET:=0;
	//PWM_Y9_SET:=0;
	//PWM_Y7_SET_Target:=0;
	//PWM_Y9_SET_Target:=0;
	GVL_SaveEngine.PWM_Y33_SET_Target:=417;//排量110->120  下降初始排量110-120 396-378-396
	IF PWM_Y33_SET>=PWM_Y33_SET_Target THEN
		PWM_Y33_SET := PWM_Y33_SET_Target;
	END_IF
	//加入斜坡防止上提结束Y33突增制动力矩减小导致的制动掉臂
	IF(PWM_Y33_SET<PWM_Y33_SET_Target) THEN
		PWM_Y33_SET:=REAL_TO_UINT(UINT_TO_REAL(PWM_Y33_SET)+JianGE6);
	END_IF
	//PWM_Y33_SET:=396;//中位排量110->130
	//PWM_Y1_SET:=300;
	//PWM_Y2_SET:=300;
	//PWM_Y1_Target_OutPut:=0;
	//PWM_Y2_Target_OutPut:=0;

//其他动作中位置0
		DOH_Y50_1:= FALSE;
		PWM_Y21_SET:=0;
		PWM_Y22_SET:=0;
		DOH_70:=FALSE;
		DOH_73:=FALSE;
		DOH_JK2:=FALSE;
			PWM_Y12_SET:=0;
			PWM_Y14_SET:=0;
			PWM_Y61_SET:=0;
			PWM_Y11_SET:=0;
			PWM_Y13_SET:=0;
			PWM_Y60_SET:=0;
			PWM_Y41_SET:=0;
			PWM_Y42_SET:=0;	
			PWM_Y59_SET:=0;	
		PWM_Y23_SET:=0;
		PWM_Y24_SET:=0;
		PWM_Y17_SET:=0;
		PWM_Y18_SET:=0;
  //Y39 40执行
	(*主泵卸荷阀控制*)
	PWM_Y39_SET_Target:=0;
	PWM_Y40_SET_Target:=0;
	RAMP19(
	IN:=WORD_TO_INT(PWM_Y39_SET_Target), 
	ASCEND:= R_RAMP_xiehe, 
	DESCEND:= F_RAMP_xiehe, 
	TIMEBASE:=TIMEBASE_xiehe , 
	RESET:=FALSE , 
	OUT=>(PWM_Y39_SET_Target1));
	IF(PWM_Y39_SET_Target1>=400) THEN
	Curve_input:=TO_UINT(PWM_Y39_SET_Target1 - 400);
	IF(Curve_input>900) THEN
		Curve_input:=900;
	END_IF
	curve19(input:=REAL_TO_UINT(UINT_TO_REAL(Curve_input)*72.8),Zero:=FALSE,Full:=FALSE,
		   PAR_Progression:=Curve_Par1,OutputEnable:=TRUE);
	PWM_Y39_SET:=PAR_Valve1_NegFull + REAL_TO_UINT(UINT_TO_REAL(curve19.Output)/72.8);
	ELSE
	PWM_Y39_SET:=0;
	END_IF


RAMP20(
	IN:=WORD_TO_INT(PWM_Y40_SET_Target), 
	ASCEND:= R_RAMP_xiehe, 
	DESCEND:= F_RAMP_xiehe, 
	TIMEBASE:=TIMEBASE_xiehe , 
	RESET:=FALSE , 
	OUT=>(PWM_Y40_SET_Target1));
IF(PWM_Y40_SET_Target1>=400) THEN
	Curve_input:=TO_UINT(PWM_Y40_SET_Target1 - 400);
	IF(Curve_input>900) THEN
		Curve_input:=900;
	END_IF
	curve20(input:=REAL_TO_UINT(UINT_TO_REAL(Curve_input)*72.8),Zero:=FALSE,Full:=FALSE,
		   PAR_Progression:=Curve_Par1,OutputEnable:=TRUE);
	PWM_Y40_SET:=PAR_Valve1_NegFull + REAL_TO_UINT(UINT_TO_REAL(curve20.Output)/72.8);
ELSE
	PWM_Y40_SET:=0;
END_IF
	
IF(PWM_Y39_SET>1300)THEN
	PWM_Y39_SET :=1300;
END_IF
IF(PWM_Y40_SET>1300)THEN
	PWM_Y40_SET :=1300;
END_IF

IF(PWM_Y39_SET<=300)THEN
	PWM_Y39_SET :=0;
END_IF
IF(PWM_Y40_SET<=300)THEN
	PWM_Y40_SET :=0;
END_IF
	(*卸荷动作缓冲*)
	//PWM_Y39_SET_Target1:=0;
	//PWM_Y40_SET_Target1:=0;
	//PWM_Y40_SET:=0;
	//PWM_Y39_SET:=0;

	
    P25_Flag:=FALSE;
    P27_Flag:=FALSE;
	P29_Flag:=FALSE; 
	P31_Flag:=FALSE;        


(*

	  (*主泵功率控制*)	
	//区分发动机转速
	IF EngineSpeedTarget<=1080 THEN SPEED_CASE:=1;
	ELSIF EngineSpeedTarget>1080 AND EngineSpeedTarget<=1300 THEN SPEED_CASE:=2;
	ELSIF EngineSpeedTarget>1300 AND EngineSpeedTarget<=1520 THEN SPEED_CASE:=3;
	ELSIF EngineSpeedTarget>1520 AND EngineSpeedTarget<=1680 THEN SPEED_CASE:=4;
	ELSIF EngineSpeedTarget>1680 AND EngineSpeedTarget<=1820 THEN SPEED_CASE:=5;
	ELSIF EngineSpeedTarget>1820 THEN SPEED_CASE:=6;;END_IF
	//不同转速下的发动机最大功率
	CASE SPEED_CASE OF
	1:  Enginer_Power:=135;
	2:  Enginer_Power:=174;
	3:  Enginer_Power:=200;
	4:  Enginer_Power:=230;
	5:  Enginer_Power:=250;
	6:  Enginer_Power:=261;
	END_CASE
	//不同转速下的压力值
	IF(CANO_Fubeng_Press<100)THEN
		CASE SPEED_CASE OF
		1:MainPump_Pressure_Taget:=MainPump_Pressure_Taget1000;
		2:MainPump_Pressure_Taget:=MainPump_Pressure_Taget1200-ECO_Press_Target1200;
		3:MainPump_Pressure_Taget:=MainPump_Pressure_Taget1450-ECO_Press_Target1400;
		4:MainPump_Pressure_Taget:=MainPump_Pressure_Taget1600-ECO_Press_Target1600;
		5:MainPump_Pressure_Taget:=MainPump_Pressure_Taget1750-ECO_Press_Target1800;
		6:MainPump_Pressure_Taget:=MainPump_Pressure_Taget1900-ECO_Press_Target1900;
		END_CASE
	ELSE
		CASE SPEED_CASE OF
		1:MainPump_Pressure_Taget:=MainPump_Pressure_Taget1000;
		2:MainPump_Pressure_Taget:=MainPump_Pressure_Taget1200;
		3:MainPump_Pressure_Taget:=MainPump_Pressure_Taget1450;
		4:MainPump_Pressure_Taget:=MainPump_Pressure_Taget1600;
		5:MainPump_Pressure_Taget:=MainPump_Pressure_Taget1750;
		6:MainPump_Pressure_Taget:=MainPump_Pressure_Taget1900;
		END_CASE		
	END_IF
	
	MainPump_Pressure:=CANO_MainPUMP_Press1+CANO_MainPUMP_Press2;
	//消除滤波
	MainPump_Pressure_Subtract:= UINT_TO_INT(MainPump_Pressure-MainPump_Pressure_last1);
	//大范围波动
	IF MainPump_Pressure_Subtract>240 OR MainPump_Pressure_Subtract<-240 THEN
		Subtract:=TRUE;
	ELSE
		Subtract:=FALSE;	
	END_IF
		TIME_LvBo4(IN:=Subtract,PT:=T#500MS);
		
	IF(TIME_LvBo4.Q) AND (NOT Joyx_change_bool) AND (CANO_MainPUMP_Press1>210) THEN 
			MainPump_Pressure_ChangeBool1:=TRUE;
	END_IF
		TIME_LvBo1(IN:=MainPump_Pressure_ChangeBool1,PT:=T#2S);
	IF(TIME_LvBo1.Q) THEN
		MainPump_Pressure_ChangeBool1 :=FALSE;
	END_IF
	
	IF(MainPump_Pressure_ChangeBool1) AND (MainPump_Pressure>MainPump_Pressure_last1) THEN 
		MainPump_Pressure_last1:=MainPump_Pressure;
	END_IF
	
	//小范围波动
	IF (NOT MainPump_Pressure_ChangeBool1) THEN
		IF(MainPump_Pressure_Subtract>30 OR MainPump_Pressure_Subtract<-30)THEN 
			MainPump_Pressure_ChangeBool:=TRUE;
		ELSE
			MainPump_Pressure_ChangeBool:=FALSE;
		END_IF
	
		TIME_LvBo2(IN:=MainPump_Pressure_ChangeBool,PT:=T#1S);
		IF(TIME_LvBo2.Q )THEN
			MainPump_Pressure_last1:=MainPump_Pressure;
		END_IF	
	END_IF
	
	
	IF PowerHead_move AND NOT(MainWinch_move) THEN
			JianGE2:=0.005;
			JianGE1:=3;
	ELSE
		IF(EngineSpeedTarget>1000 AND EngineSpeedTarget<1300)THEN
			JianGE2:=0.005;
			JianGE1:=1;
		ELSE
			JianGE2:=0.008;
			JianGE1:=1.7;	
		END_IF
	END_IF
	
	IF( CANI_ECOSwitch) THEN
		ECO_Press_Target1200 := 40;
		ECO_Press_Target1400 := 60;
		ECO_Press_Target1600 := 75;
		ECO_Press_Target1800 := 75;
		ECO_Press_Target1900 := 75;	
	ELSE
		ECO_Press_Target1200 := 0;
		ECO_Press_Target1400 := 0;
		ECO_Press_Target1600 := 0;
		ECO_Press_Target1800 := 0;
		ECO_Press_Target1900 := 0;
	END_IF
		
	IF MainPump_Pressure_last1>MainPump_Pressure_Taget THEN
		Pressure_Coe_Taget:=UINT_TO_REAL(MainPump_Pressure_Taget)/UINT_TO_REAL(MainPump_Pressure_last1);(*压力系数*)
	ELSE
		Pressure_Coe_Taget:=1;
	END_IF
	
	TIME_100ms(in:=NOT TIME_100ms.Q,pt:=T#10MS);
	
	IF(Pressure_Coe_Taget>Pressure_Coe) THEN
		IF(TIME_100ms.Q) THEN
			Pressure_Coe := Pressure_Coe + JianGE2;
		END_IF
	ELSE
		Pressure_Coe := Pressure_Coe_Taget;
	END_IF
	
	IF MainPump_Pressure_last1>MainPump_Pressure_Taget  THEN
		IF(PWM_Y1_Target>=PAR_Y1_1_NegFull)THEN
			PWM_Y1_Target_OutPut:=REAL_TO_UINT(UINT_TO_REAL(PWM_Y1_Target-PAR_Y1_1_NegFull)*Pressure_Coe+PAR_Y1_1_NegFull);
		END_IF
		IF(PWM_Y2_Target>=PAR_Y1_1_NegFull)THEN
			PWM_Y2_Target_OutPut:=REAL_TO_UINT(UINT_TO_REAL(PWM_Y2_Target-PAR_Y1_1_NegFull)*Pressure_Coe+PAR_Y1_1_NegFull);
		END_IF
	ELSE
		PWM_Y1_Target_OutPut:=PWM_Y1_Target;
		PWM_Y2_Target_OutPut:=PWM_Y2_Target;
	END_IF
	
	IF(EngineSpeedTarget>CANO_SPEED AND CANO_SPEED>400)THEN
		EngineSpeedSub:=EngineSpeedTarget - CANO_SPEED;
	ELSE
		EngineSpeedSub:=0;
	END_IF
	
	IF(PWM_Y1_Target_OutPut<300)THEN PWM_Y1_Target_OutPut:=300;END_IF	
	IF(PWM_Y2_Target_OutPut<300)THEN PWM_Y2_Target_OutPut:=300;END_IF
	IF LeftMove_move OR RightMove_move THEN
		yanchi1:=TRUE;
	ELSE
		yanchi1:=FALSE;		
	END_IF
	yanchi_ton1(IN:=yanchi1 , PT:=T#300MS);
	IF (NOT yanchi1) OR yanchi_ton1.Q THEN
		RAMP15_IN:=PWM_Y1_Target_OutPut;
		RAMP16_IN:=PWM_Y2_Target_OutPut;
	ELSE
		RAMP15_IN:=PAR_Y1_1_NegFull;
		RAMP16_IN:=PAR_Y1_1_NegFull;
	END_IF
	
	RAMP15(
		IN:=UINT_TO_INT(RAMP15_IN), 
		ASCEND:= R_RAMP_3, 
		DESCEND:= F_RAMP_3, 
		TIMEBASE:=TIMEBASE_3 , 
		RESET:=FALSE , 
		OUT=>(PWM_Y1_SET));
		
	RAMP16(
		IN:=UINT_TO_INT(RAMP16_IN), 
		ASCEND:= R_RAMP_3, 
		DESCEND:= F_RAMP_3, 
		TIMEBASE:=TIMEBASE_3 , 
		RESET:=FALSE , 
		OUT=>(PWM_Y2_SET));
	IF PWM_Y1_SET<TO_INT(PAR_Y1_1_NegFull )THEN
		PWM_Y1_SET:=TO_INT(PAR_Y1_1_NegFull);
	END_IF
	IF PWM_Y2_SET<TO_INT(PAR_Y1_1_NegFull )THEN
		PWM_Y2_SET:=TO_INT(PAR_Y1_1_NegFull);
	END_IF
	IF(PWM_Y1_SET>1000) THEN
		PWM_Y1_SET := 300;
	END_IF
	IF(PWM_Y2_SET>1000) THEN
		PWM_Y2_SET := 300;
	END_IF		
*)


//IF(PWM_Y1_Target_OutPut<300)THEN PWM_Y1_Target_OutPut:=300;END_IF	
//IF(PWM_Y2_Target_OutPut<300)THEN PWM_Y2_Target_OutPut:=300;END_IF
RAMP15_IN:=300;
RAMP16_IN:=300;
(*
RAMP15(
	IN:=UINT_TO_INT(RAMP15_IN), 
	ASCEND:= 300, 
	DESCEND:= 400, 
	TIMEBASE:=T#1000MS , 
	RESET:=FALSE , 
	OUT=>(PWM_Y1_SET));
(******减斜坡300->400*****)	
RAMP16(
	IN:=UINT_TO_INT(RAMP16_IN), 
	ASCEND:= 300, 
	DESCEND:= 400, 
	TIMEBASE:=T#1000MS , 
	RESET:=FALSE , 
	OUT=>(PWM_Y2_SET));
*)
	CASE SPEED_CASE OF
                1:F_RAMP_pump:=1500; R_RAMP_pump:=100;                  
                2: 		IF MainWinch_move AND (JiaYa_move OR CANO_JiayaPressure>80)  THEN    //3泵同时起压时，降低主泵的加载速度，避免掉速熄火
                                F_RAMP_pump:=1500; R_RAMP_pump:=100;
                        ELSE
                                F_RAMP_pump:=1500; R_RAMP_pump:=100;//从200降
                                IF  PWM_JOYY_L_UP>10 THEN
                                 F_RAMP_pump:=1500; R_RAMP_pump:=200;
                                END_IF
                        END_IF            
                3:
                        IF MainWinch_move AND (JiaYa_move OR CANO_JiayaPressure>80)  THEN    //3泵同时起压时，降低主泵的加载速度，避免掉速熄火
                                F_RAMP_pump:=1500; R_RAMP_pump:=150;
                        ELSE
                                F_RAMP_pump:=1500; R_RAMP_pump:=TO_INT(PAR_NegFull_y);
                                IF  PWM_JOYY_L_UP>10 THEN
                                 F_RAMP_pump:=1500; R_RAMP_pump:=300;
                                END_IF
                        END_IF                
                4:
                        IF MainWinch_move AND (JiaYa_move OR CANO_JiayaPressure>80)  THEN
                                F_RAMP_pump:=1500; R_RAMP_pump:=150;
                        ELSE
                                F_RAMP_pump:=1500; R_RAMP_pump:=TO_INT(PAR_PosFull_y);//从200降
                                IF  PWM_JOYY_L_UP>10 THEN
                                 F_RAMP_pump:=1500; R_RAMP_pump:=300;
                                END_IF
                        END_IF                                
                5:
                        IF MainWinch_move AND (JiaYa_move OR CANO_JiayaPressure>80)  THEN
                                F_RAMP_pump:=1500; R_RAMP_pump:=200;
                        ELSE
                                F_RAMP_pump:=1500; R_RAMP_pump:=TO_INT(PAR_Zero_y);
                                IF  PWM_JOYY_L_UP>10 THEN
                                 F_RAMP_pump:=1500; R_RAMP_pump:=300;
                                END_IF
                        END_IF                        
                6:		IF MainWinch_move AND (JiaYa_move OR CANO_JiayaPressure>80)  THEN
                                F_RAMP_pump:=1500; R_RAMP_pump:=200;
                        ELSE
                                F_RAMP_pump:=1500; R_RAMP_pump:=200;
                                IF  PWM_JOYY_L_UP>10 THEN
                                 F_RAMP_pump:=1500; R_RAMP_pump:=300;
                                END_IF
                        END_IF	
	END_CASE
(******斜坡增步长300 斜坡降步长300->400*****)	
RAMP15(
	IN:=UINT_TO_INT(RAMP15_IN), 
	ASCEND:= R_RAMP_pump, 
	DESCEND:= 1500, 
	TIMEBASE:=T#1000MS , 
	RESET:=FALSE , 
	OUT=>(PWM_Y1_SET));
(******减斜坡300->400*****)	
RAMP16(
	IN:=UINT_TO_INT(RAMP16_IN), 
	ASCEND:= R_RAMP_pump, 
	DESCEND:= 1500, 
	TIMEBASE:=T#1000MS , 
	RESET:=FALSE , 
	OUT=>(PWM_Y2_SET));

END_PROGRAM

// StandardPLC/Application/SaveEngine/SaveEngineMode_5
PROGRAM SaveEngineMode_5
VAR

END_VAR


(*******************节能控制阀主阀主泵输出执行**************************)
	
//ELSIF(GVL_SaveEngine.SaveEngineMode=5)THEN//泄压模式
	GVL_SaveEngine.Y72OutPutState:=0;
	GVL_SaveEngine.Y71OutPutState:=1;
	DOH_Y56:=TRUE;//
	Y73:=FALSE;	
	IF(UIGroupVoltage0<2000 OR UIGroupVoltage1<2000 OR UIGroupVoltage2<2000 
	   OR UIGroupVoltage3<2000 OR UIGroupVoltage4<2000 OR UIGroupVoltage5<2000) THEN
		reset111:=TRUE;
	ELSE
		reset111:=FALSE;
	END_IF
	(*冷却风扇控制*)
	IF NOT CANI_ColdFunSwitch  THEN
		IF(CANO_Hyd_Tem>60)THEN
			PWM_Y49_SET := PAR_ValveD_NegFull;
		END_IF
		
		IF(CANO_Hyd_Tem<60)THEN
			PWM_Y49_SET := 0;		
		END_IF
	ELSE
		PWM_Y49_SET := PAR_ValveD_NegFull;
	END_IF
	

	IF(UIGroupVoltage0<2000 OR UIGroupVoltage1<2000 OR UIGroupVoltage2<2000 
	   OR UIGroupVoltage3<2000 OR UIGroupVoltage4<2000 OR UIGroupVoltage5<2000) THEN
		reset111:=TRUE;
	ELSE
		reset111:=FALSE;
	END_IF

END_PROGRAM

// StandardPLC/Application/SaveEngine/SaveEngineMode_6
PROGRAM SaveEngineMode_6
VAR
	PressLvBo_TON:TON;
	PressLvBo_TON1: TON;
	PressLvBo_TON2: TON;
	PressLvBo_TON3: TON;
END_VAR


(*******************节能控制阀主阀主泵输出执行**************************)
	
//ELSIF(GVL_SaveEngine.SaveEngineMode=6)THEN  //上升微动模式	
	GVL_SaveEngine.Y72OutPutState:=0;
	GVL_SaveEngine.Y71OutPutState:=0;
	DOH_Y56:=FALSE;
		Y73:=FALSE;	
	PWM_Y1_Target:=REAL_TO_UINT(UINT_TO_REAL(PWM_JOYY_L_DOWN)/1000*(PAR_Y1_PosFull-PAR_Y1_NegFull)+PAR_Y1_NegFull);
	PWM_Y2_Target:=REAL_TO_UINT(UINT_TO_REAL(PWM_JOYY_L_DOWN)/1000*(PAR_Y2_PosFull-PAR_Y2_NegFull)+PAR_Y2_NegFull);
	PWM_Y7_SET_Target:=REAL_TO_UINT(UINT_TO_REAL(PWM_JOYY_L_DOWN)/1000*(PAR_Valve1_PosFull-PAR_Valve2_NegFull)+PAR_Valve2_NegFull);
	PWM_Y9_SET_Target:=REAL_TO_UINT(UINT_TO_REAL(PWM_JOYY_L_DOWN)/1000*(PAR_Valve2_PosFull-PAR_Valve2_NegFull)+PAR_Valve2_NegFull);
	PWM_Y8_SET_Target:=300;
	PWM_Y10_SET_Target:=300;	
	
	(*电控马达主卷变量控制*)
	PressLvBo_TON(IN:=CANO_ZhuJuanPressure>310,PT:=T#300MS);
	PressLvBo_TON1(IN:=CANO_ZhuJuanPressure>290 AND CANO_ZhuJuanPressure<=310,PT:=T#300MS);
	PressLvBo_TON2(IN:=CANO_ZhuJuanPressure>270 AND CANO_ZhuJuanPressure<=290,PT:=T#300MS);
	PressLvBo_TON3(IN:=CANO_ZhuJuanPressure>250 AND CANO_ZhuJuanPressure<=270,PT:=T#300MS);
	IF(CANO_ZhuJuanPressure>310 AND PressLvBo_TON.Q) OR P31_Flag THEN
        PWM_Y33_SET_Target :=230;   //排量200
        P31_Flag:=TRUE;
        IF (CANO_ZhuJuanPressure<270) THEN
                P31_Flag:=FALSE;        
        END_IF
	ELSIF(CANO_ZhuJuanPressure>290 AND PressLvBo_TON1.Q) OR P29_Flag THEN   
        PWM_Y33_SET_Target :=267;   //排量180
        P29_Flag:=TRUE; 
        IF (CANO_ZhuJuanPressure<250) THEN
                P29_Flag:=FALSE; 
        END_IF
	ELSIF(CANO_ZhuJuanPressure>270 AND PressLvBo_TON2.Q) OR P27_Flag THEN   
        PWM_Y33_SET_Target :=304;  //排量160
        P27_Flag:=TRUE;
        IF (CANO_ZhuJuanPressure<230) THEN
                P27_Flag:=FALSE; 
        END_IF
	ELSIF(CANO_ZhuJuanPressure>250 AND PressLvBo_TON3.Q) OR P25_Flag THEN //压力小于270   
        PWM_Y33_SET_Target :=340;  //排量140
        P25_Flag:=TRUE; 
        IF (CANO_ZhuJuanPressure<210) THEN
                P25_Flag:=FALSE; 
        END_IF
	ELSE //(CANO_ZhuJuanPressure<=250) THEN
        PWM_Y33_SET_Target :=370;
	END_IF
(*	
	IF BiaoZHI_MainWinchUp THEN  //单主卷下放370马达电流
 		PWM_Y33_SET_Target:=370;
	END_IF
*)
	IF PWM_Y33_SET>=PWM_Y33_SET_Target THEN
		PWM_Y33_SET := PWM_Y33_SET_Target;
	END_IF
	IF(PWM_Y33_SET<PWM_Y33_SET_Target) THEN
		PWM_Y33_SET:=REAL_TO_UINT(UINT_TO_REAL(PWM_Y33_SET)+JianGE6);
	END_IF
	IF DIL_SQ3 THEN
		PWM_Y33_SET:=0;
	END_IF	
	

(*主泵功率控制*)

//区分发动机转速
MainPump_Pressure_Taget1450:=PAR_NegFull_x;
MainPump_Pressure_Taget1600:=PAR_PosFull_x;
MainPump_Pressure_Taget1750:=PAR_Zero_x;
IF EngineSpeedTarget<=1080 THEN SPEED_CASE:=1;
ELSIF EngineSpeedTarget>1080 AND EngineSpeedTarget<=1300 THEN SPEED_CASE:=2;
ELSIF EngineSpeedTarget>1300 AND EngineSpeedTarget<=1520 THEN SPEED_CASE:=3;
ELSIF EngineSpeedTarget>1520 AND EngineSpeedTarget<=1680 THEN SPEED_CASE:=4;
ELSIF EngineSpeedTarget>1680 AND EngineSpeedTarget<=1820 THEN SPEED_CASE:=5;
ELSIF EngineSpeedTarget>1820 THEN SPEED_CASE:=6;;END_IF
//不同转速下的发动机最大功率*)
CASE SPEED_CASE OF
1:  Enginer_Power:=135;
2:  Enginer_Power:=174;
3:  Enginer_Power:=200;
4:  Enginer_Power:=230;
5:  Enginer_Power:=250;
6:  Enginer_Power:=261;
END_CASE
//不同转速下的压力值
IF(CANO_Fubeng_Press>100)THEN
	CASE SPEED_CASE OF
	1:MainPump_Pressure_Taget:=MainPump_Pressure_Taget1000-HELIU_Press_Target1000;
	2:MainPump_Pressure_Taget:=MainPump_Pressure_Taget1200-HELIU_Press_Target1200;
	3:MainPump_Pressure_Taget:=MainPump_Pressure_Taget1450-HELIU_Press_Target1400;
	4:MainPump_Pressure_Taget:=MainPump_Pressure_Taget1600-HELIU_Press_Target1600;
	5:MainPump_Pressure_Taget:=MainPump_Pressure_Taget1750-HELIU_Press_Target1800;
	6:MainPump_Pressure_Taget:=MainPump_Pressure_Taget1900-HELIU_Press_Target1900;
	END_CASE
ELSE
	CASE SPEED_CASE OF
	1:MainPump_Pressure_Taget:=MainPump_Pressure_Taget1000;
	2:MainPump_Pressure_Taget:=MainPump_Pressure_Taget1200;
	3:MainPump_Pressure_Taget:=MainPump_Pressure_Taget1450;
	4:MainPump_Pressure_Taget:=MainPump_Pressure_Taget1600;
	5:MainPump_Pressure_Taget:=MainPump_Pressure_Taget1750;
	6:MainPump_Pressure_Taget:=MainPump_Pressure_Taget1900;
	END_CASE		
END_IF

IF( CANI_ECOSwitch) THEN
	CASE SPEED_CASE OF
	1:MainPump_Pressure_Taget:=MainPump_Pressure_Taget1000-ECO_Press_Target1000;
	2:MainPump_Pressure_Taget:=MainPump_Pressure_Taget1200-ECO_Press_Target1200;
	3:MainPump_Pressure_Taget:=MainPump_Pressure_Taget1450-ECO_Press_Target1400;
	4:MainPump_Pressure_Taget:=MainPump_Pressure_Taget1600-ECO_Press_Target1600;
	5:MainPump_Pressure_Taget:=MainPump_Pressure_Taget1750-ECO_Press_Target1800;
	6:MainPump_Pressure_Taget:=MainPump_Pressure_Taget1900-ECO_Press_Target1900;
	END_CASE
END_IF
MainPump_Pressure:=CANO_MainPUMP_Press1+CANO_MainPUMP_Press2;
//消除滤波
MainPump_Pressure_Subtract:= UINT_TO_INT(MainPump_Pressure-MainPump_Pressure_last1);


//大范围波动
IF MainPump_Pressure_Subtract>270 OR MainPump_Pressure_Subtract<-270 THEN
	Subtract:=TRUE;
ELSE
	Subtract:=FALSE;	
END_IF
	TIME_LvBo4(IN:=Subtract,PT:=T#10MS);
	
IF(TIME_LvBo4.Q) AND (CANO_MainPUMP_Press1>210) THEN 
		MainPump_Pressure_ChangeBool1:=TRUE;
END_IF
	TIME_LvBo1(IN:=MainPump_Pressure_ChangeBool1,PT:=T#2S);
IF(TIME_LvBo1.Q) THEN
	MainPump_Pressure_ChangeBool1 :=FALSE;
END_IF

IF(MainPump_Pressure_ChangeBool1) AND (MainPump_Pressure>MainPump_Pressure_last1) THEN 
	MainPump_Pressure_last1:=MainPump_Pressure;
END_IF

//小范围波动
t_powertime:=TO_TIME(PAR_DeadBand_x);
IF (NOT MainPump_Pressure_ChangeBool1) THEN
	IF(MainPump_Pressure_Subtract>40 OR MainPump_Pressure_Subtract<-40)THEN 
		MainPump_Pressure_ChangeBool:=TRUE;
	ELSE
		MainPump_Pressure_ChangeBool:=FALSE;
	END_IF

	TIME_LvBo2(IN:=MainPump_Pressure_ChangeBool,PT:=t_powertime);
	IF(TIME_LvBo2.Q )THEN
		MainPump_Pressure_last1:=MainPump_Pressure;
	END_IF	
END_IF


IF PowerHead_move AND NOT(MainWinch_move) THEN
		JianGE2:=0.005;
ELSE
	IF(EngineSpeedTarget>1000 AND EngineSpeedTarget<1300)THEN
		JianGE2:=0.005;
	ELSE
		JianGE2:=0.005;
	END_IF
END_IF
	
IF MainPump_Pressure_last1>MainPump_Pressure_Taget THEN
	Pressure_Coe_Taget:=UINT_TO_REAL(MainPump_Pressure_Taget)/UINT_TO_REAL(MainPump_Pressure_last1);(*压力系数*)
ELSE
	Pressure_Coe_Taget:=1;
END_IF
Pressure_Coe := Pressure_Coe_Taget;

IF MainPump_Pressure_last1>MainPump_Pressure_Taget  THEN
	IF(PWM_Y1_Target>=PAR_Y1_1_NegFull)THEN
		PWM_Y1_Target_OutPut:=REAL_TO_UINT(UINT_TO_REAL(PWM_Y1_Target-PAR_Y1_1_NegFull)*Pressure_Coe+PAR_Y1_1_NegFull);
	END_IF
	IF(PWM_Y2_Target>=PAR_Y1_1_NegFull)THEN
		PWM_Y2_Target_OutPut:=REAL_TO_UINT(UINT_TO_REAL(PWM_Y2_Target-PAR_Y1_1_NegFull)*Pressure_Coe+PAR_Y1_1_NegFull);
	END_IF
ELSE
	PWM_Y1_Target_OutPut:=PWM_Y1_Target;
	PWM_Y2_Target_OutPut:=PWM_Y2_Target;
END_IF

//PWM_Y1_Target_OutPut:=PWM_Y1_Target;
//PWM_Y2_Target_OutPut:=PWM_Y2_Target;
IF(EngineSpeedTarget>CANO_SPEED AND CANO_SPEED>400)THEN
	EngineSpeedSub:=EngineSpeedTarget - CANO_SPEED;
ELSE
	EngineSpeedSub:=0;
END_IF

IF(PWM_Y1_Target_OutPut<300)THEN PWM_Y1_Target_OutPut:=300;END_IF	
IF(PWM_Y2_Target_OutPut<300)THEN PWM_Y2_Target_OutPut:=300;END_IF

RAMP15_IN:=PWM_Y1_Target_OutPut;
RAMP16_IN:=PWM_Y2_Target_OutPut;
(*
IF MainWinch_move  OR  LeftMove_move OR RightMove_move THEN  
	TIMEBASE_pump:=T#1000MS;
	TIMEBASE_xiehe:=T#500MS;
ELSE
	TIMEBASE_pump:=T#400MS;
	TIMEBASE_xiehe:=T#200MS;
END_IF
t_PowerHead_move(IN:= MainWinch_move,PT:=T#2S);
IF t_PowerHead_move.Q THEN
	F_RAMP_pump:=x_t_PowerHead_move;
	R_RAMP_pump:=x2_t_PowerHead_move;
ELSE
	F_RAMP_pump:=1000;
	R_RAMP_pump:=300;
END_IF
*)
(*
RAMP15(
	IN:=UINT_TO_INT(RAMP15_IN), 
	ASCEND:= 300, 
	DESCEND:= 400, 
	TIMEBASE:=T#1000MS , 
	RESET:=FALSE , 
	OUT=>(PWM_Y1_SET));
	
RAMP16(
	IN:=UINT_TO_INT(RAMP16_IN), 
	ASCEND:= 300, 
	DESCEND:= 400, 
	TIMEBASE:=T#1000MS , 
	RESET:=FALSE , 
	OUT=>(PWM_Y2_SET));
*)
	CASE SPEED_CASE OF
                1:F_RAMP_pump:=1500; R_RAMP_pump:=100;                  
                2: 		IF MainWinch_move AND (JiaYa_move OR CANO_JiayaPressure>80)  THEN    //3泵同时起压时，降低主泵的加载速度，避免掉速熄火
                                F_RAMP_pump:=1500; R_RAMP_pump:=100;
                        ELSE
                                F_RAMP_pump:=1500; R_RAMP_pump:=100;//从200降
                                IF  PWM_JOYY_L_UP>10 THEN
                                 F_RAMP_pump:=1500; R_RAMP_pump:=200;
                                END_IF
                        END_IF            
                3:
                        IF MainWinch_move AND (JiaYa_move OR CANO_JiayaPressure>80)  THEN    //3泵同时起压时，降低主泵的加载速度，避免掉速熄火
                                F_RAMP_pump:=1500; R_RAMP_pump:=150;
                        ELSE
                                F_RAMP_pump:=1500; R_RAMP_pump:=TO_INT(PAR_NegFull_y);
                                IF  PWM_JOYY_L_UP>10 THEN
                                 F_RAMP_pump:=1500; R_RAMP_pump:=300;
                                END_IF
                        END_IF                
                4:
                        IF MainWinch_move AND (JiaYa_move OR CANO_JiayaPressure>80)  THEN
                                F_RAMP_pump:=1500; R_RAMP_pump:=150;
                        ELSE
                                F_RAMP_pump:=1500; R_RAMP_pump:=TO_INT(PAR_PosFull_y);//从200降
                                IF  PWM_JOYY_L_UP>10 THEN
                                 F_RAMP_pump:=1500; R_RAMP_pump:=300;
                                END_IF
                        END_IF                                
                5:
                        IF MainWinch_move AND (JiaYa_move OR CANO_JiayaPressure>80)  THEN
                                F_RAMP_pump:=1500; R_RAMP_pump:=200;
                        ELSE
                                F_RAMP_pump:=1500; R_RAMP_pump:=TO_INT(PAR_Zero_y);
                                IF  PWM_JOYY_L_UP>10 THEN
                                 F_RAMP_pump:=1500; R_RAMP_pump:=300;
                                END_IF
                        END_IF                        
                6:		IF MainWinch_move AND (JiaYa_move OR CANO_JiayaPressure>80)  THEN
                                F_RAMP_pump:=1500; R_RAMP_pump:=200;
                        ELSE
                                F_RAMP_pump:=1500; R_RAMP_pump:=200;
                                IF  PWM_JOYY_L_UP>10 THEN
                                 F_RAMP_pump:=1500; R_RAMP_pump:=300;
                                END_IF
                        END_IF	
	END_CASE
(******斜坡增步长300 斜坡降步长300->400*****)	
RAMP15(
	IN:=UINT_TO_INT(RAMP15_IN), 
	ASCEND:= R_RAMP_pump, 
	DESCEND:= 1500, 
	TIMEBASE:=T#1000MS , 
	RESET:=FALSE , 
	OUT=>(PWM_Y1_SET));
(******减斜坡300->400*****)	
RAMP16(
	IN:=UINT_TO_INT(RAMP16_IN), 
	ASCEND:= R_RAMP_pump, 
	DESCEND:= 1500, 
	TIMEBASE:=T#1000MS , 
	RESET:=FALSE , 
	OUT=>(PWM_Y2_SET));

IF (NOT Rotation_move) AND (NOT MainWinch_move) AND (NOT PowerHead_move)
		AND (NOT JiaYa_move) AND (NOT ViceWinch_move)
		AND (NOT LeftMove_move) AND (NOT RightMove_move)  THEN
	PWM_Y1_Target:=0;
	PWM_Y2_Target:=0;
END_IF


IF PWM_Y1_SET<TO_INT(PAR_Y1_1_NegFull )THEN
	PWM_Y1_SET:=TO_INT(PAR_Y1_1_NegFull);
END_IF

IF PWM_Y2_SET<TO_INT(PAR_Y1_1_NegFull )THEN
	PWM_Y2_SET:=TO_INT(PAR_Y1_1_NegFull);
END_IF

IF(PWM_Y1_SET>1000) THEN
	PWM_Y1_SET := 300;
END_IF

IF(PWM_Y2_SET>1000) THEN
	PWM_Y2_SET := 300;
END_IF	
  //Y7 8 9 10处理	
		IF(PWM_Y8_SET<1000  AND  PWM_Y8_SET>=900)THEN    //主卷下放斜坡值
				F_RAMP_mainwinch_down:=200;
			
			ELSIF(PWM_Y8_SET<900)THEN
				F_RAMP_mainwinch_down:=400;
			ELSE
				F_RAMP_mainwinch_down:=400;
			END_IF
			
		IF(PWM_Y7_SET<1000  AND  PWM_Y7_SET>=900)THEN  //主卷上提斜坡值
				F_RAMP_mainwinch_down:=300;
		ELSIF(PWM_Y7_SET<900  )THEN
				F_RAMP_mainwinch_down:=200;
		ELSE
				F_RAMP_mainwinch_down:=400;
		END_IF
			
	RAMP7(
		IN:=WORD_TO_INT(PWM_Y7_SET_Target), 
		ASCEND:= R_RAMP_mainwinch, 
		DESCEND:= F_RAMP_mainwinch_up, 
		TIMEBASE:=TIMEBASE_mainwinch , 
		RESET:=FALSE , 
		OUT=>(PWM_Y7_SET_Target1));
	IF(PWM_Y7_SET_Target1>=400) THEN
		Curve_input:=TO_UINT(PWM_Y7_SET_Target1 - 400);
		IF(Curve_input>900) THEN
			Curve_input:=900;
		END_IF
		curve7(input:=REAL_TO_UINT(UINT_TO_REAL(Curve_input)*72.8),Zero:=FALSE,Full:=FALSE,
			   PAR_Progression:=Curve_Par,OutputEnable:=TRUE);
		PWM_Y7_SET:=PAR_Valve1_NegFull + REAL_TO_UINT(UINT_TO_REAL(curve7.Output)/72.8);
	ELSE
		PWM_Y7_SET:=0;
	END_IF
	
	
	RAMP8(
		IN:=WORD_TO_INT(PWM_Y8_SET_Target), 
		ASCEND:= R_RAMP_mainwinch, 
		DESCEND:= F_RAMP_mainwinch_down, 
		TIMEBASE:=TIMEBASE_mainwinch , 
		RESET:=FALSE , 
		OUT=>(PWM_Y8_SET_Target1));
	IF(PWM_Y8_SET_Target1>=400) THEN
		Curve_input:=TO_UINT(PWM_Y8_SET_Target1 - 400);
		IF(Curve_input>900) THEN
			Curve_input:=900;
		END_IF
		curve8(input:=REAL_TO_UINT(UINT_TO_REAL(Curve_input)*72.8),Zero:=FALSE,Full:=FALSE,
			   PAR_Progression:=Curve_Par,OutputEnable:=TRUE);
		PWM_Y8_SET:=PAR_Valve1_NegFull + REAL_TO_UINT(UINT_TO_REAL(curve8.Output)/72.8);
	ELSE
		PWM_Y8_SET:=0;
	END_IF
	
	
	RAMP9(
		IN:=WORD_TO_INT(PWM_Y9_SET_Target), 
		ASCEND:= R_RAMP_mainwinch, 
		DESCEND:= F_RAMP_mainwinch_up, 
		TIMEBASE:=TIMEBASE_mainwinch , 
		RESET:=FALSE , 
		OUT=>(PWM_Y9_SET_Target1));
	IF(PWM_Y9_SET_Target1>=400) THEN
		Curve_input:=TO_UINT(PWM_Y9_SET_Target1 - 400);
		IF(Curve_input>900) THEN
			Curve_input:=900;
		END_IF
		curve9(input:=REAL_TO_UINT(UINT_TO_REAL(Curve_input)*72.8),Zero:=FALSE,Full:=FALSE,
			   PAR_Progression:=Curve_Par,OutputEnable:=TRUE);
		PWM_Y9_SET:=PAR_Valve1_NegFull + REAL_TO_UINT(UINT_TO_REAL(curve9.Output)/72.8);
	ELSE
		PWM_Y9_SET:=0;
	END_IF
	
	RAMP10(
		IN:=WORD_TO_INT(PWM_Y10_SET_Target), 
		ASCEND:= R_RAMP_mainwinch, 
		DESCEND:= F_RAMP_mainwinch_down, 
		TIMEBASE:=TIMEBASE_mainwinch , 
		RESET:=FALSE , 
		OUT=>(PWM_Y10_SET_Target1));
	IF(PWM_Y10_SET_Target1>=400) THEN
		Curve_input:=TO_UINT(PWM_Y10_SET_Target1 - 400);
		IF(Curve_input>900) THEN
			Curve_input:=900;
		END_IF
		curve10(input:=REAL_TO_UINT(UINT_TO_REAL(Curve_input)*72.8),Zero:=FALSE,Full:=FALSE,
			   PAR_Progression:=Curve_Par,OutputEnable:=TRUE);
		PWM_Y10_SET:=PAR_Valve1_NegFull + REAL_TO_UINT(UINT_TO_REAL(curve10.Output)/72.8);
	ELSE
		PWM_Y10_SET:=0;
	END_IF
    //Y7 8 9 10范围限制
	IF(PWM_Y7_SET>1300)THEN
		PWM_Y7_SET :=1300;
	END_IF
	IF(PWM_Y8_SET>1300)THEN
		PWM_Y8_SET :=1300;
	END_IF
	IF(PWM_Y9_SET>1300)THEN
		PWM_Y9_SET :=1300;
	END_IF
	IF(PWM_Y10_SET>1300)THEN
		PWM_Y10_SET :=1300;
	END_IF
	
	IF(PWM_Y7_SET<=300)THEN
		PWM_Y7_SET :=0;
	END_IF
	IF(PWM_Y8_SET<=300)THEN
		PWM_Y8_SET :=0;
	END_IF
	IF(PWM_Y9_SET<=300)THEN
		PWM_Y9_SET :=0;
	END_IF
	IF(PWM_Y10_SET<=300)THEN
		PWM_Y10_SET :=0;
	END_IF
	(*主泵卸荷阀控制*)
		PWM_Y39_SET_Target:=MAX(PWM_Y8_SET_Target,PWM_Y7_SET_Target);
		PWM_Y40_SET_Target:=MAX(PWM_Y9_SET_Target,PWM_Y10_SET_Target);
	(*卸荷动作缓冲*)
RAMP19(
	IN:=WORD_TO_INT(PWM_Y39_SET_Target), 
	ASCEND:= R_RAMP_xiehe, 
	DESCEND:= F_RAMP_xiehe, 
	TIMEBASE:=TIMEBASE_xiehe , 
	RESET:=FALSE , 
	OUT=>(PWM_Y39_SET_Target1));
IF(PWM_Y39_SET_Target1>=400) THEN
	Curve_input:=TO_UINT(PWM_Y39_SET_Target1 - 400);
	IF(Curve_input>900) THEN
		Curve_input:=900;
	END_IF
	curve19(input:=REAL_TO_UINT(UINT_TO_REAL(Curve_input)*72.8),Zero:=FALSE,Full:=FALSE,
		   PAR_Progression:=Curve_Par1,OutputEnable:=TRUE);
	PWM_Y39_SET:=PAR_Valve1_NegFull + REAL_TO_UINT(UINT_TO_REAL(curve19.Output)/72.8);
ELSE
	PWM_Y39_SET:=0;
END_IF


RAMP20(
	IN:=WORD_TO_INT(PWM_Y40_SET_Target), 
	ASCEND:= R_RAMP_xiehe, 
	DESCEND:= F_RAMP_xiehe, 
	TIMEBASE:=TIMEBASE_xiehe , 
	RESET:=FALSE , 
	OUT=>(PWM_Y40_SET_Target1));
IF(PWM_Y40_SET_Target1>=400) THEN
	Curve_input:=TO_UINT(PWM_Y40_SET_Target1 - 400);
	IF(Curve_input>900) THEN
		Curve_input:=900;
	END_IF
	curve20(input:=REAL_TO_UINT(UINT_TO_REAL(Curve_input)*72.8),Zero:=FALSE,Full:=FALSE,
		   PAR_Progression:=Curve_Par1,OutputEnable:=TRUE);
	PWM_Y40_SET:=PAR_Valve1_NegFull + REAL_TO_UINT(UINT_TO_REAL(curve20.Output)/72.8);
ELSE
	PWM_Y40_SET:=0;
END_IF
	
IF(PWM_Y39_SET>1300)THEN
	PWM_Y39_SET :=1300;
END_IF
IF(PWM_Y40_SET>1300)THEN
	PWM_Y40_SET :=1300;
END_IF

IF(PWM_Y39_SET<=300)THEN
	PWM_Y39_SET :=0;
END_IF
IF(PWM_Y40_SET<=300)THEN
	PWM_Y40_SET :=0;
END_IF

END_PROGRAM

// StandardPLC/Application/SaveEngine/SaveEngineMode_7
PROGRAM SaveEngineMode_7
VAR

END_VAR


(*******************节能控制阀主阀主泵输出执行**************************)
//ELSIF(GVL_SaveEngine.SaveEngineMode=7)THEN  //下放微动模式	,先按常规的写
	//Y72先关，200ms后 Y71关闭
	//GVL_SaveEngine.Y72OutPutState:=0;
	//GVL_SaveEngine.Y71OutPutState:=0;
	GVL_SaveEngine.Y72OutPutState:=0;
	IF Mode7Timer>0 THEN
		GVL_SaveEngine.Y71OutPutState:=0;
	END_IF
	
	DOH_Y56:=FALSE;
	Y73:=FALSE;	
	PWM_Y1_Target:=REAL_TO_UINT(UINT_TO_REAL(PWM_JOYY_L_UP)/1000*(PAR_Y1_PosFull-PAR_Y1_NegFull)+PAR_Y1_NegFull);
	PWM_Y2_Target:=REAL_TO_UINT(UINT_TO_REAL(PWM_JOYY_L_UP)/1000*(PAR_Y2_PosFull-PAR_Y2_NegFull)+PAR_Y2_NegFull);
	PWM_Y8_SET_Target:=REAL_TO_UINT(UINT_TO_REAL(PWM_JOYY_L_UP)/1000*(PAR_Valve1_PosFull-PAR_Valve1_NegFull)+PAR_Valve1_NegFull);
	PWM_Y10_SET_Target:=REAL_TO_UINT(UINT_TO_REAL(PWM_JOYY_L_UP)/1000*(PAR_Valve2_PosFull-PAR_Valve2_NegFull)+PAR_Valve2_NegFull);
	PWM_Y7_SET_Target:=0;
	PWM_Y9_SET_Target:=0;
	PWM_Y33_SET_Target:=417; //  下降初始排量125-120  370-378-396
  //Y33输出处理
	IF PWM_Y33_SET>=PWM_Y33_SET_Target THEN
	PWM_Y33_SET := PWM_Y33_SET_Target;
	END_IF
		
	IF(PWM_Y33_SET<PWM_Y33_SET_Target) THEN
		PWM_Y33_SET:=REAL_TO_UINT(UINT_TO_REAL(PWM_Y33_SET)+JianGE6);
	END_IF
	
	IF DIL_SQ3 THEN
		PWM_Y33_SET:=0;
	END_IF
	
(*主泵功率控制*)

//区分发动机转速
MainPump_Pressure_Taget1450:=PAR_NegFull_x;
MainPump_Pressure_Taget1600:=PAR_PosFull_x;
MainPump_Pressure_Taget1750:=PAR_Zero_x;
IF EngineSpeedTarget<=1080 THEN SPEED_CASE:=1;
ELSIF EngineSpeedTarget>1080 AND EngineSpeedTarget<=1300 THEN SPEED_CASE:=2;
ELSIF EngineSpeedTarget>1300 AND EngineSpeedTarget<=1520 THEN SPEED_CASE:=3;
ELSIF EngineSpeedTarget>1520 AND EngineSpeedTarget<=1680 THEN SPEED_CASE:=4;
ELSIF EngineSpeedTarget>1680 AND EngineSpeedTarget<=1820 THEN SPEED_CASE:=5;
ELSIF EngineSpeedTarget>1820 THEN SPEED_CASE:=6;;END_IF
//不同转速下的发动机最大功率*)
CASE SPEED_CASE OF
1:  Enginer_Power:=135;
2:  Enginer_Power:=174;
3:  Enginer_Power:=200;
4:  Enginer_Power:=230;
5:  Enginer_Power:=250;
6:  Enginer_Power:=261;
END_CASE
//不同转速下的压力值
IF(CANO_Fubeng_Press>100)THEN
	CASE SPEED_CASE OF
	1:MainPump_Pressure_Taget:=MainPump_Pressure_Taget1000-HELIU_Press_Target1000;
	2:MainPump_Pressure_Taget:=MainPump_Pressure_Taget1200-HELIU_Press_Target1200;
	3:MainPump_Pressure_Taget:=MainPump_Pressure_Taget1450-HELIU_Press_Target1400;
	4:MainPump_Pressure_Taget:=MainPump_Pressure_Taget1600-HELIU_Press_Target1600;
	5:MainPump_Pressure_Taget:=MainPump_Pressure_Taget1750-HELIU_Press_Target1800;
	6:MainPump_Pressure_Taget:=MainPump_Pressure_Taget1900-HELIU_Press_Target1900;
	END_CASE
ELSE
	CASE SPEED_CASE OF
	1:MainPump_Pressure_Taget:=MainPump_Pressure_Taget1000;
	2:MainPump_Pressure_Taget:=MainPump_Pressure_Taget1200;
	3:MainPump_Pressure_Taget:=MainPump_Pressure_Taget1450;
	4:MainPump_Pressure_Taget:=MainPump_Pressure_Taget1600;
	5:MainPump_Pressure_Taget:=MainPump_Pressure_Taget1750;
	6:MainPump_Pressure_Taget:=MainPump_Pressure_Taget1900;
	END_CASE		
END_IF

IF( CANI_ECOSwitch) THEN
	CASE SPEED_CASE OF
	1:MainPump_Pressure_Taget:=MainPump_Pressure_Taget1000-ECO_Press_Target1000;
	2:MainPump_Pressure_Taget:=MainPump_Pressure_Taget1200-ECO_Press_Target1200;
	3:MainPump_Pressure_Taget:=MainPump_Pressure_Taget1450-ECO_Press_Target1400;
	4:MainPump_Pressure_Taget:=MainPump_Pressure_Taget1600-ECO_Press_Target1600;
	5:MainPump_Pressure_Taget:=MainPump_Pressure_Taget1750-ECO_Press_Target1800;
	6:MainPump_Pressure_Taget:=MainPump_Pressure_Taget1900-ECO_Press_Target1900;
	END_CASE
END_IF
MainPump_Pressure:=CANO_MainPUMP_Press1+CANO_MainPUMP_Press2;
//消除滤波
MainPump_Pressure_Subtract:= UINT_TO_INT(MainPump_Pressure-MainPump_Pressure_last1);


//大范围波动
IF MainPump_Pressure_Subtract>270 OR MainPump_Pressure_Subtract<-270 THEN
	Subtract:=TRUE;
ELSE
	Subtract:=FALSE;	
END_IF
	TIME_LvBo4(IN:=Subtract,PT:=T#10MS);
	
IF(TIME_LvBo4.Q) AND (CANO_MainPUMP_Press1>210) THEN 
		MainPump_Pressure_ChangeBool1:=TRUE;
END_IF
	TIME_LvBo1(IN:=MainPump_Pressure_ChangeBool1,PT:=T#2S);
IF(TIME_LvBo1.Q) THEN
	MainPump_Pressure_ChangeBool1 :=FALSE;
END_IF

IF(MainPump_Pressure_ChangeBool1) AND (MainPump_Pressure>MainPump_Pressure_last1) THEN 
	MainPump_Pressure_last1:=MainPump_Pressure;
END_IF

//小范围波动
t_powertime:=TO_TIME(PAR_DeadBand_x);
IF (NOT MainPump_Pressure_ChangeBool1) THEN
	IF(MainPump_Pressure_Subtract>40 OR MainPump_Pressure_Subtract<-40)THEN 
		MainPump_Pressure_ChangeBool:=TRUE;
	ELSE
		MainPump_Pressure_ChangeBool:=FALSE;
	END_IF

	TIME_LvBo2(IN:=MainPump_Pressure_ChangeBool,PT:=t_powertime);
	IF(TIME_LvBo2.Q )THEN
		MainPump_Pressure_last1:=MainPump_Pressure;
	END_IF	
END_IF


IF PowerHead_move AND NOT(MainWinch_move) THEN
		JianGE2:=0.005;
ELSE
	IF(EngineSpeedTarget>1000 AND EngineSpeedTarget<1300)THEN
		JianGE2:=0.005;
	ELSE
		JianGE2:=0.005;
	END_IF
END_IF

IF MainPump_Pressure_last1>MainPump_Pressure_Taget THEN
	Pressure_Coe_Taget:=UINT_TO_REAL(MainPump_Pressure_Taget)/UINT_TO_REAL(MainPump_Pressure_last1);(*压力系数*)
ELSE
	Pressure_Coe_Taget:=1;
END_IF
Pressure_Coe := Pressure_Coe_Taget;


IF MainPump_Pressure_last1>MainPump_Pressure_Taget  THEN
	IF(PWM_Y1_Target>=PAR_Y1_1_NegFull)THEN
		PWM_Y1_Target_OutPut:=REAL_TO_UINT(UINT_TO_REAL(PWM_Y1_Target-PAR_Y1_1_NegFull)*Pressure_Coe+PAR_Y1_1_NegFull);
	END_IF
	IF(PWM_Y2_Target>=PAR_Y1_1_NegFull)THEN
		PWM_Y2_Target_OutPut:=REAL_TO_UINT(UINT_TO_REAL(PWM_Y2_Target-PAR_Y1_1_NegFull)*Pressure_Coe+PAR_Y1_1_NegFull);
	END_IF
ELSE
	PWM_Y1_Target_OutPut:=PWM_Y1_Target;
	PWM_Y2_Target_OutPut:=PWM_Y2_Target;
END_IF

//PWM_Y1_Target_OutPut:=PWM_Y1_Target; 
//PWM_Y2_Target_OutPut:=PWM_Y2_Target;

IF(EngineSpeedTarget>CANO_SPEED AND CANO_SPEED>400)THEN
	EngineSpeedSub:=EngineSpeedTarget - CANO_SPEED;
ELSE
	EngineSpeedSub:=0;
END_IF

IF(PWM_Y1_Target_OutPut<300)THEN PWM_Y1_Target_OutPut:=300;END_IF	
IF(PWM_Y2_Target_OutPut<300)THEN PWM_Y2_Target_OutPut:=300;END_IF

RAMP15_IN:=PWM_Y1_Target_OutPut;
RAMP16_IN:=PWM_Y2_Target_OutPut;
(*
RAMP15(
	IN:=UINT_TO_INT(RAMP15_IN), 
	ASCEND:= 900, 
	DESCEND:= 400, 
	TIMEBASE:=T#1000MS , 
	RESET:=FALSE , 
	OUT=>(PWM_Y1_SET));
(*****反弹 增加斜坡值  让主泵电流快速加***)	
RAMP16(
	IN:=UINT_TO_INT(RAMP16_IN), 
	ASCEND:= 900, 
	DESCEND:= 400, 
	TIMEBASE:=T#1000MS , 
	RESET:=FALSE , 
	OUT=>(PWM_Y2_SET));
*)
	CASE SPEED_CASE OF
                1:F_RAMP_pump:=1500; R_RAMP_pump:=100;                  
                2: 		IF MainWinch_move AND (JiaYa_move OR CANO_JiayaPressure>80)  THEN    //3泵同时起压时，降低主泵的加载速度，避免掉速熄火
                                F_RAMP_pump:=1500; R_RAMP_pump:=100;
                        ELSE
                                F_RAMP_pump:=1500; R_RAMP_pump:=100;//从200降
                                IF  PWM_JOYY_L_UP>10 THEN
                                 F_RAMP_pump:=1500; R_RAMP_pump:=200;
                                END_IF
                        END_IF            
                3:
                        IF MainWinch_move AND (JiaYa_move OR CANO_JiayaPressure>80)  THEN    //3泵同时起压时，降低主泵的加载速度，避免掉速熄火
                                F_RAMP_pump:=1500; R_RAMP_pump:=150;
                        ELSE
                                F_RAMP_pump:=1500; R_RAMP_pump:=TO_INT(PAR_NegFull_y);
                                IF  PWM_JOYY_L_UP>10 THEN
                                 F_RAMP_pump:=1500; R_RAMP_pump:=300;
                                END_IF
                        END_IF                
                4:
                        IF MainWinch_move AND (JiaYa_move OR CANO_JiayaPressure>80)  THEN
                                F_RAMP_pump:=1500; R_RAMP_pump:=150;
                        ELSE
                                F_RAMP_pump:=1500; R_RAMP_pump:=TO_INT(PAR_PosFull_y);//从200降
                                IF  PWM_JOYY_L_UP>10 THEN
                                 F_RAMP_pump:=1500; R_RAMP_pump:=300;
                                END_IF
                        END_IF                                
                5:
                        IF MainWinch_move AND (JiaYa_move OR CANO_JiayaPressure>80)  THEN
                                F_RAMP_pump:=1500; R_RAMP_pump:=200;
                        ELSE
                                F_RAMP_pump:=1500; R_RAMP_pump:=TO_INT(PAR_Zero_y);
                                IF  PWM_JOYY_L_UP>10 THEN
                                 F_RAMP_pump:=1500; R_RAMP_pump:=300;
                                END_IF
                        END_IF                        
                6:		IF MainWinch_move AND (JiaYa_move OR CANO_JiayaPressure>80)  THEN
                                F_RAMP_pump:=1500; R_RAMP_pump:=200;
                        ELSE
                                F_RAMP_pump:=1500; R_RAMP_pump:=200;
                                IF  PWM_JOYY_L_UP>10 THEN
                                 F_RAMP_pump:=1500; R_RAMP_pump:=300;
                                END_IF
                        END_IF
	END_CASE

(******斜坡增步长300 斜坡降步长300->400*****)	
RAMP15(
	IN:=UINT_TO_INT(RAMP15_IN), 
	ASCEND:= 900, 
	DESCEND:= 1500, 
	TIMEBASE:=T#1000MS , 
	RESET:=FALSE , 
	OUT=>(PWM_Y1_SET));
(******减斜坡300->400*****)	
RAMP16(
	IN:=UINT_TO_INT(RAMP16_IN), 
	ASCEND:= 900, 
	DESCEND:= 1500, 
	TIMEBASE:=T#1000MS , 
	RESET:=FALSE , 
	OUT=>(PWM_Y2_SET));
	
	
IF (NOT Rotation_move) AND (NOT MainWinch_move) AND (NOT PowerHead_move)
		AND (NOT JiaYa_move) AND (NOT ViceWinch_move)
		AND (NOT LeftMove_move) AND (NOT RightMove_move)  THEN
	PWM_Y1_Target:=0;
	PWM_Y2_Target:=0;
END_IF


IF PWM_Y1_SET<TO_INT(PAR_Y1_1_NegFull )THEN
	PWM_Y1_SET:=TO_INT(PAR_Y1_1_NegFull);
END_IF

IF PWM_Y2_SET<TO_INT(PAR_Y1_1_NegFull )THEN
	PWM_Y2_SET:=TO_INT(PAR_Y1_1_NegFull);
END_IF

IF(PWM_Y1_SET>1000) THEN
	PWM_Y1_SET := 300;
END_IF

IF(PWM_Y2_SET>1000) THEN
	PWM_Y2_SET := 300;
END_IF	
  //Y7 8 9 10处理	
		IF(PWM_Y8_SET<1000  AND  PWM_Y8_SET>=900)THEN    //主卷下放斜坡值
				F_RAMP_mainwinch_down:=200;
			
			ELSIF(PWM_Y8_SET<900)THEN
				F_RAMP_mainwinch_down:=400;
			ELSE
				F_RAMP_mainwinch_down:=400;
			END_IF
			
		IF(PWM_Y7_SET<1000  AND  PWM_Y7_SET>=900)THEN  //主卷上提斜坡值
				F_RAMP_mainwinch_down:=300;
		ELSIF(PWM_Y7_SET<900  )THEN
				F_RAMP_mainwinch_down:=200;
		ELSE
				F_RAMP_mainwinch_down:=400;
		END_IF
			
	RAMP7(
		IN:=WORD_TO_INT(PWM_Y7_SET_Target), 
		ASCEND:= R_RAMP_mainwinch, 
		DESCEND:= F_RAMP_mainwinch_up, 
		TIMEBASE:=TIMEBASE_mainwinch , 
		RESET:=FALSE , 
		OUT=>(PWM_Y7_SET_Target1));
	IF(PWM_Y7_SET_Target1>=400) THEN
		Curve_input:=TO_UINT(PWM_Y7_SET_Target1 - 400);
		IF(Curve_input>900) THEN
			Curve_input:=900;
		END_IF
		curve7(input:=REAL_TO_UINT(UINT_TO_REAL(Curve_input)*72.8),Zero:=FALSE,Full:=FALSE,
			   PAR_Progression:=Curve_Par,OutputEnable:=TRUE);
		PWM_Y7_SET:=PAR_Valve1_NegFull + REAL_TO_UINT(UINT_TO_REAL(curve7.Output)/72.8);
	ELSE
		PWM_Y7_SET:=0;
	END_IF
	
	
	RAMP8(
		IN:=WORD_TO_INT(PWM_Y8_SET_Target), 
		ASCEND:= R_RAMP_mainwinch, 
		DESCEND:= F_RAMP_mainwinch_down, 
		TIMEBASE:=TIMEBASE_mainwinch , 
		RESET:=FALSE , 
		OUT=>(PWM_Y8_SET_Target1));
	IF(PWM_Y8_SET_Target1>=400) THEN
		Curve_input:=TO_UINT(PWM_Y8_SET_Target1 - 400);
		IF(Curve_input>900) THEN
			Curve_input:=900;
		END_IF
		curve8(input:=REAL_TO_UINT(UINT_TO_REAL(Curve_input)*72.8),Zero:=FALSE,Full:=FALSE,
			   PAR_Progression:=Curve_Par,OutputEnable:=TRUE);
		PWM_Y8_SET:=PAR_Valve1_NegFull + REAL_TO_UINT(UINT_TO_REAL(curve8.Output)/72.8);
	ELSE
		PWM_Y8_SET:=0;
	END_IF
	
	
	RAMP9(
		IN:=WORD_TO_INT(PWM_Y9_SET_Target), 
		ASCEND:= R_RAMP_mainwinch, 
		DESCEND:= F_RAMP_mainwinch_up, 
		TIMEBASE:=TIMEBASE_mainwinch , 
		RESET:=FALSE , 
		OUT=>(PWM_Y9_SET_Target1));
	IF(PWM_Y9_SET_Target1>=400) THEN
		Curve_input:=TO_UINT(PWM_Y9_SET_Target1 - 400);
		IF(Curve_input>900) THEN
			Curve_input:=900;
		END_IF
		curve9(input:=REAL_TO_UINT(UINT_TO_REAL(Curve_input)*72.8),Zero:=FALSE,Full:=FALSE,
			   PAR_Progression:=Curve_Par,OutputEnable:=TRUE);
		PWM_Y9_SET:=PAR_Valve1_NegFull + REAL_TO_UINT(UINT_TO_REAL(curve9.Output)/72.8);
	ELSE
		PWM_Y9_SET:=0;
	END_IF
	
	RAMP10(
		IN:=WORD_TO_INT(PWM_Y10_SET_Target), 
		ASCEND:= R_RAMP_mainwinch, 
		DESCEND:= F_RAMP_mainwinch_down, 
		TIMEBASE:=TIMEBASE_mainwinch , 
		RESET:=FALSE , 
		OUT=>(PWM_Y10_SET_Target1));
	IF(PWM_Y10_SET_Target1>=400) THEN
		Curve_input:=TO_UINT(PWM_Y10_SET_Target1 - 400);
		IF(Curve_input>900) THEN
			Curve_input:=900;
		END_IF
		curve10(input:=REAL_TO_UINT(UINT_TO_REAL(Curve_input)*72.8),Zero:=FALSE,Full:=FALSE,
			   PAR_Progression:=Curve_Par,OutputEnable:=TRUE);
		PWM_Y10_SET:=PAR_Valve1_NegFull + REAL_TO_UINT(UINT_TO_REAL(curve10.Output)/72.8);
	ELSE
		PWM_Y10_SET:=0;
	END_IF
    //Y7 8 9 10范围限制
	IF(PWM_Y7_SET>1300)THEN
		PWM_Y7_SET :=1300;
	END_IF
	IF(PWM_Y8_SET>1300)THEN
		PWM_Y8_SET :=1300;
	END_IF
	IF(PWM_Y9_SET>1300)THEN
		PWM_Y9_SET :=1300;
	END_IF
	IF(PWM_Y10_SET>1300)THEN
		PWM_Y10_SET :=1300;
	END_IF
	
	IF(PWM_Y7_SET<=300)THEN
		PWM_Y7_SET :=0;
	END_IF
	IF(PWM_Y8_SET<=300)THEN
		PWM_Y8_SET :=0;
	END_IF
	IF(PWM_Y9_SET<=300)THEN
		PWM_Y9_SET :=0;
	END_IF
	IF(PWM_Y10_SET<=300)THEN
		PWM_Y10_SET :=0;
	END_IF
	(*主泵卸荷阀控制*)
		PWM_Y39_SET_Target:=MAX(PWM_Y8_SET_Target,PWM_Y7_SET_Target);
		PWM_Y40_SET_Target:=MAX(PWM_Y9_SET_Target,PWM_Y10_SET_Target);
	(*卸荷动作缓冲*)
RAMP19(
	IN:=WORD_TO_INT(PWM_Y39_SET_Target), 
	ASCEND:= R_RAMP_xiehe, 
	DESCEND:= F_RAMP_xiehe, 
	TIMEBASE:=TIMEBASE_xiehe , 
	RESET:=FALSE , 
	OUT=>(PWM_Y39_SET_Target1));
IF(PWM_Y39_SET_Target1>=400) THEN
	Curve_input:=TO_UINT(PWM_Y39_SET_Target1 - 400);
	IF(Curve_input>900) THEN
		Curve_input:=900;
	END_IF
	curve19(input:=REAL_TO_UINT(UINT_TO_REAL(Curve_input)*72.8),Zero:=FALSE,Full:=FALSE,
		   PAR_Progression:=Curve_Par1,OutputEnable:=TRUE);
	PWM_Y39_SET:=PAR_Valve1_NegFull + REAL_TO_UINT(UINT_TO_REAL(curve19.Output)/72.8);
ELSE
	PWM_Y39_SET:=0;
END_IF


RAMP20(
	IN:=WORD_TO_INT(PWM_Y40_SET_Target), 
	ASCEND:= R_RAMP_xiehe, 
	DESCEND:= F_RAMP_xiehe, 
	TIMEBASE:=TIMEBASE_xiehe , 
	RESET:=FALSE , 
	OUT=>(PWM_Y40_SET_Target1));
IF(PWM_Y40_SET_Target1>=400) THEN
	Curve_input:=TO_UINT(PWM_Y40_SET_Target1 - 400);
	IF(Curve_input>900) THEN
		Curve_input:=900;
	END_IF
	curve20(input:=REAL_TO_UINT(UINT_TO_REAL(Curve_input)*72.8),Zero:=FALSE,Full:=FALSE,
		   PAR_Progression:=Curve_Par1,OutputEnable:=TRUE);
	PWM_Y40_SET:=PAR_Valve1_NegFull + REAL_TO_UINT(UINT_TO_REAL(curve20.Output)/72.8);
ELSE
	PWM_Y40_SET:=0;
END_IF
	
IF(PWM_Y39_SET>1300)THEN
	PWM_Y39_SET :=1300;
END_IF
IF(PWM_Y40_SET>1300)THEN
	PWM_Y40_SET :=1300;
END_IF

IF(PWM_Y39_SET<=300)THEN
	PWM_Y39_SET :=0;
END_IF
IF(PWM_Y40_SET<=300)THEN
	PWM_Y40_SET :=0;
END_IF

END_PROGRAM

// StandardPLC/Application/SaveEngine/SaveEngineMode_8
PROGRAM SaveEngineMode_8
VAR

	TON1: TON;
	TON2: TON;
	AI_PM2Pre_Flag1: BOOL;
	AI_PM2Pre_Flag3: BOOL;
	PM2Pre_Rtrig1: R_TRIG;
	PM2Pre_Rtrig3: R_TRIG;
	Mod1CasePWM_Y1:UINT;
	A: UINT;
	B: UINT;
END_VAR


(*******************节能控制阀主阀主泵输出执行**************************)
	
//ELSIF(GVL_SaveEngine.SaveEngineMode=8)THEN  //下放收满能模式 ,先按常规执行
	//Y72先关，200ms后 Y71关闭
	//GVL_SaveEngine.Y72OutPutState:=0;
	//GVL_SaveEngine.Y71OutPutState:=0;
	GVL_SaveEngine.Y72OutPutState:=0;
	IF Mode8Timer>0 THEN
		GVL_SaveEngine.Y71OutPutState:=0;
	END_IF
	DOH_Y56:=FALSE;
	Y73:=FALSE;	
	//PWM_Y1_Target:=REAL_TO_UINT(UINT_TO_REAL(PWM_JOYY_L_UP)/1000*(PAR_Y1_PosFull-PAR_Y1_NegFull)+PAR_Y1_NegFull);
	//PWM_Y2_Target:=REAL_TO_UINT(UINT_TO_REAL(PWM_JOYY_L_UP)/1000*(PAR_Y2_PosFull-PAR_Y2_NegFull)+PAR_Y2_NegFull);
	//PWM_Y8_SET_Target:=REAL_TO_UINT(UINT_TO_REAL(PWM_JOYY_L_UP)/1000*(PAR_Valve1_PosFull-PAR_Valve1_NegFull)+PAR_Valve1_NegFull);
	//PWM_Y10_SET_Target:=REAL_TO_UINT(UINT_TO_REAL(PWM_JOYY_L_UP)/1000*(PAR_Valve2_PosFull-PAR_Valve2_NegFull)+PAR_Valve2_NegFull);
	//PWM_Y7_SET_Target:=0;
	//PWM_Y9_SET_Target:=0;
	//PWM_Y33_SET_Target:=370;
  //Y33输出处理
 //M2>6MPa持续1s Y33>230,每过1s Y33+18,排量减10，至Y33>450
 //M2<3MPa持续200ms且马达排量>80,每200ms Y33-18,排量+10  
  	TON1(IN:=NOT TON1.Q AND GVL_SaveEngine.AI_PM2Pre<30 ,PT:=T#200MS);
	TON2(IN:=NOT TON2.Q AND GVL_SaveEngine.AI_PM2Pre>=60 ,PT:=T#1S);
	IF TON2.Q AND GVL_SaveEngine.PWM_Y33_SET_Target<500 THEN
		AI_PM2Pre_Flag1:=TRUE;
	ELSE
		AI_PM2Pre_Flag1:=FALSE;
	END_IF
	IF GVL_SaveEngine.PWM_Y33_SET_Target>=230 AND TON1.Q  THEN
		AI_PM2Pre_Flag3:=TRUE;
	ELSE
		AI_PM2Pre_Flag3:=FALSE;
	END_IF

	PM2Pre_Rtrig1(CLK:=AI_PM2Pre_Flag1);
	PM2Pre_Rtrig3(CLK:=AI_PM2Pre_Flag3);

	IF(PM2Pre_Rtrig1.Q)THEN
		//A:=A+1;
		GVL_SaveEngine.PWM_Y33_SET_Target:=GVL_SaveEngine.PWM_Y33_SET_Target+17;
		AI_PM2Pre_Flag1:=FALSE;
	END_IF
	
	IF(PM2Pre_Rtrig3.Q)THEN
		//B:=B+1;
		GVL_SaveEngine.PWM_Y33_SET_Target:=GVL_SaveEngine.PWM_Y33_SET_Target-17;
		AI_PM2Pre_Flag3:=FALSE;
	END_IF
	GVL_SaveEngine.PWM_Y33_SET_Target:=LIMIT(417,GVL_SaveEngine.PWM_Y33_SET_Target,465);
	PWM_Y33_SET := GVL_SaveEngine.PWM_Y33_SET_Target;//去掉原有坡度执行防止干扰
	
	(*IF PWM_Y33_SET>=PWM_Y33_SET_Target THEN
	PWM_Y33_SET := PWM_Y33_SET_Target;
	END_IF
		
	IF(PWM_Y33_SET<PWM_Y33_SET_Target) THEN
		PWM_Y33_SET:=REAL_TO_UINT(UINT_TO_REAL(PWM_Y33_SET)+JianGE6);
	END_IF
	*)
	IF DIL_SQ3 THEN
		PWM_Y33_SET:=0;
	END_IF
	//和1模式一样，根据档位设定目标电流，以及主卷排量计算主泵最大电流
		CASE AI_ECM2_Flag OF
			1: Mod1CasePWM_Y1:=REAL_TO_UINT(362.5+47.8*30/1100*(600-PWM_Y33_SET)/1.85)+40;
			2: Mod1CasePWM_Y1:=REAL_TO_UINT(362.5+47.8*42/1200*(600-PWM_Y33_SET)/1.85)+40;
			3: Mod1CasePWM_Y1:=REAL_TO_UINT(362.5+47.8*55/1450*(600-PWM_Y33_SET)/1.85)+40;
			4: Mod1CasePWM_Y1:=REAL_TO_UINT(362.5+47.8*62/1500*(600-PWM_Y33_SET)/1.85)+120;//调速  40->55 20230418
			5: Mod1CasePWM_Y1:=REAL_TO_UINT(362.5+47.8*68/1500*(600-PWM_Y33_SET)/1.85)+120;//0-75
			6: Mod1CasePWM_Y1:=REAL_TO_UINT(362.5+47.8*72/1500*(600-PWM_Y33_SET)/1.85)+120;//-20-75
		END_CASE
		
	PWM_Y1_Target:=REAL_TO_UINT(UINT_TO_REAL(PWM_JOYY_L_UP)/1000*(Mod1CasePWM_Y1-PAR_Y1_NegFull)+PAR_Y1_NegFull);
	PWM_Y2_Target:=REAL_TO_UINT(UINT_TO_REAL(PWM_JOYY_L_UP)/1000*(Mod1CasePWM_Y1-PAR_Y2_NegFull)+PAR_Y2_NegFull);
	IF PWM_Y1_Target>700 THEN 
		PWM_Y1_Target:=700;
	END_IF
	IF PWM_Y2_Target>700 THEN 
		PWM_Y2_Target:=700;
	END_IF																																																																																																																																																																																																																																																																																																																																																																																																																																																																																																																																																																																																																																																																																																																																																																																																																																																																																																																																																																																																																																																																																																																																																																																																																																																																																																																																																																																																																																																																																																																																																																																																																																																																																																																																																																																																																																																																																																																																																																																																																																																																																																																																																																																																																																																																																																																																																																																																																																																																																																																																																																																																																																																																																																																																																																																																																																																																																																																																																																																																																																																																																																																																																																																																																																																																																																																																																																																																																																																																																																																																																																																																																																																																																																																																																																																																																																																																																																																																																																																																																																																																																																																																																																																																																																																																									
(*	
	PWM_Y1_SET:=UINT_TO_INT(PWM_Y1_Target);
	PWM_Y2_SET:=UINT_TO_INT(PWM_Y2_Target);
*)	

	
(*主泵功率控制*)

//区分发动机转速
MainPump_Pressure_Taget1450:=PAR_NegFull_x;
MainPump_Pressure_Taget1600:=PAR_PosFull_x;
MainPump_Pressure_Taget1750:=PAR_Zero_x;
IF EngineSpeedTarget<=1080 THEN SPEED_CASE:=1;
ELSIF EngineSpeedTarget>1080 AND EngineSpeedTarget<=1300 THEN SPEED_CASE:=2;
ELSIF EngineSpeedTarget>1300 AND EngineSpeedTarget<=1520 THEN SPEED_CASE:=3;
ELSIF EngineSpeedTarget>1520 AND EngineSpeedTarget<=1680 THEN SPEED_CASE:=4;
ELSIF EngineSpeedTarget>1680 AND EngineSpeedTarget<=1820 THEN SPEED_CASE:=5;
ELSIF EngineSpeedTarget>1820 THEN SPEED_CASE:=6;;END_IF
//不同转速下的发动机最大功率*)
CASE SPEED_CASE OF
1:  Enginer_Power:=135;
2:  Enginer_Power:=174;
3:  Enginer_Power:=200;
4:  Enginer_Power:=230;
5:  Enginer_Power:=250;
6:  Enginer_Power:=261;
END_CASE
//不同转速下的压力值
IF(CANO_Fubeng_Press>100)THEN
	CASE SPEED_CASE OF
	1:MainPump_Pressure_Taget:=MainPump_Pressure_Taget1000-HELIU_Press_Target1000;
	2:MainPump_Pressure_Taget:=MainPump_Pressure_Taget1200-HELIU_Press_Target1200;
	3:MainPump_Pressure_Taget:=MainPump_Pressure_Taget1450-HELIU_Press_Target1400;
	4:MainPump_Pressure_Taget:=MainPump_Pressure_Taget1600-HELIU_Press_Target1600;
	5:MainPump_Pressure_Taget:=MainPump_Pressure_Taget1750-HELIU_Press_Target1800;
	6:MainPump_Pressure_Taget:=MainPump_Pressure_Taget1900-HELIU_Press_Target1900;
	END_CASE
ELSE
	CASE SPEED_CASE OF
	1:MainPump_Pressure_Taget:=MainPump_Pressure_Taget1000;
	2:MainPump_Pressure_Taget:=MainPump_Pressure_Taget1200;
	3:MainPump_Pressure_Taget:=MainPump_Pressure_Taget1450;
	4:MainPump_Pressure_Taget:=MainPump_Pressure_Taget1600;
	5:MainPump_Pressure_Taget:=MainPump_Pressure_Taget1750;
	6:MainPump_Pressure_Taget:=MainPump_Pressure_Taget1900;
	END_CASE		
END_IF

IF( CANI_ECOSwitch) THEN
	CASE SPEED_CASE OF
	1:MainPump_Pressure_Taget:=MainPump_Pressure_Taget1000-ECO_Press_Target1000;
	2:MainPump_Pressure_Taget:=MainPump_Pressure_Taget1200-ECO_Press_Target1200;
	3:MainPump_Pressure_Taget:=MainPump_Pressure_Taget1450-ECO_Press_Target1400;
	4:MainPump_Pressure_Taget:=MainPump_Pressure_Taget1600-ECO_Press_Target1600;
	5:MainPump_Pressure_Taget:=MainPump_Pressure_Taget1750-ECO_Press_Target1800;
	6:MainPump_Pressure_Taget:=MainPump_Pressure_Taget1900-ECO_Press_Target1900;
	END_CASE
END_IF
MainPump_Pressure:=CANO_MainPUMP_Press1+CANO_MainPUMP_Press2;
//消除滤波
MainPump_Pressure_Subtract:= UINT_TO_INT(MainPump_Pressure-MainPump_Pressure_last1);


//大范围波动
IF MainPump_Pressure_Subtract>270 OR MainPump_Pressure_Subtract<-270 THEN
	Subtract:=TRUE;
ELSE
	Subtract:=FALSE;	
END_IF
	TIME_LvBo4(IN:=Subtract,PT:=T#10MS);
	
IF(TIME_LvBo4.Q) AND (CANO_MainPUMP_Press1>210) THEN 
		MainPump_Pressure_ChangeBool1:=TRUE;
END_IF
	TIME_LvBo1(IN:=MainPump_Pressure_ChangeBool1,PT:=T#2S);
IF(TIME_LvBo1.Q) THEN
	MainPump_Pressure_ChangeBool1 :=FALSE;
END_IF

IF(MainPump_Pressure_ChangeBool1) AND (MainPump_Pressure>MainPump_Pressure_last1) THEN 
	MainPump_Pressure_last1:=MainPump_Pressure;
END_IF

//小范围波动
t_powertime:=TO_TIME(PAR_DeadBand_x);
IF (NOT MainPump_Pressure_ChangeBool1) THEN
	IF(MainPump_Pressure_Subtract>40 OR MainPump_Pressure_Subtract<-40)THEN 
		MainPump_Pressure_ChangeBool:=TRUE;
	ELSE
		MainPump_Pressure_ChangeBool:=FALSE;
	END_IF

	TIME_LvBo2(IN:=MainPump_Pressure_ChangeBool,PT:=t_powertime);
	IF(TIME_LvBo2.Q )THEN
		MainPump_Pressure_last1:=MainPump_Pressure;
	END_IF	
END_IF


IF PowerHead_move AND NOT(MainWinch_move) THEN
		JianGE2:=0.005;
ELSE
	IF(EngineSpeedTarget>1000 AND EngineSpeedTarget<1300)THEN
		JianGE2:=0.005;
	ELSE
		JianGE2:=0.005;
	END_IF
END_IF

IF MainPump_Pressure_last1>MainPump_Pressure_Taget THEN
	Pressure_Coe_Taget:=UINT_TO_REAL(MainPump_Pressure_Taget)/UINT_TO_REAL(MainPump_Pressure_last1);(*压力系数*)
ELSE
	Pressure_Coe_Taget:=1;
END_IF
Pressure_Coe := Pressure_Coe_Taget;

IF MainPump_Pressure_last1>MainPump_Pressure_Taget  THEN
	IF(PWM_Y1_Target>=PAR_Y1_1_NegFull)THEN
		PWM_Y1_Target_OutPut:=REAL_TO_UINT(UINT_TO_REAL(PWM_Y1_Target-PAR_Y1_1_NegFull)*Pressure_Coe+PAR_Y1_1_NegFull);
	END_IF
	IF(PWM_Y2_Target>=PAR_Y1_1_NegFull)THEN
		PWM_Y2_Target_OutPut:=REAL_TO_UINT(UINT_TO_REAL(PWM_Y2_Target-PAR_Y1_1_NegFull)*Pressure_Coe+PAR_Y1_1_NegFull);
	END_IF
ELSE
	PWM_Y1_Target_OutPut:=PWM_Y1_Target;
	PWM_Y2_Target_OutPut:=PWM_Y2_Target;
END_IF

//PWM_Y1_Target_OutPut:=PWM_Y1_Target;
//PWM_Y2_Target_OutPut:=PWM_Y2_Target;
IF(EngineSpeedTarget>CANO_SPEED AND CANO_SPEED>400)THEN
	EngineSpeedSub:=EngineSpeedTarget - CANO_SPEED;
ELSE
	EngineSpeedSub:=0;
END_IF

IF(PWM_Y1_Target_OutPut<300)THEN PWM_Y1_Target_OutPut:=300;END_IF	
IF(PWM_Y2_Target_OutPut<300)THEN PWM_Y2_Target_OutPut:=300;END_IF

RAMP15_IN:=PWM_Y1_Target_OutPut;
RAMP16_IN:=PWM_Y2_Target_OutPut;
(*
IF MainWinch_move  OR  LeftMove_move OR RightMove_move THEN  
	TIMEBASE_pump:=T#1000MS;
	TIMEBASE_xiehe:=T#500MS;
ELSE
	TIMEBASE_pump:=T#400MS;
	TIMEBASE_xiehe:=T#200MS;
END_IF
t_PowerHead_move(IN:= MainWinch_move,PT:=T#2S);
IF t_PowerHead_move.Q THEN
	F_RAMP_pump:=x_t_PowerHead_move;
	R_RAMP_pump:=x2_t_PowerHead_move;
ELSE
	F_RAMP_pump:=1000;
	R_RAMP_pump:=300;
END_IF
*)

(*
RAMP15(
	IN:=UINT_TO_INT(RAMP15_IN), 
	ASCEND:= 300, 
	DESCEND:= 400, 
	TIMEBASE:=T#1000MS , 
	RESET:=FALSE , 
	OUT=>(PWM_Y1_SET));
	
RAMP16(
	IN:=UINT_TO_INT(RAMP16_IN), 
	ASCEND:= 300, 
	DESCEND:= 400, 
	TIMEBASE:=T#1000MS , 
	RESET:=FALSE , 
	OUT=>(PWM_Y2_SET));
*)
	CASE SPEED_CASE OF
                1:F_RAMP_pump:=1500; R_RAMP_pump:=100;                  
                2: 		IF MainWinch_move AND (JiaYa_move OR CANO_JiayaPressure>80)  THEN    //3泵同时起压时，降低主泵的加载速度，避免掉速熄火
                                F_RAMP_pump:=1500; R_RAMP_pump:=100;
                        ELSE
                                F_RAMP_pump:=1500; R_RAMP_pump:=100;//从200降
                                IF  PWM_JOYY_L_UP>10 THEN
                                 F_RAMP_pump:=1500; R_RAMP_pump:=200;
                                END_IF
                        END_IF            
                3:
                        IF MainWinch_move AND (JiaYa_move OR CANO_JiayaPressure>80)  THEN    //3泵同时起压时，降低主泵的加载速度，避免掉速熄火
                                F_RAMP_pump:=1500; R_RAMP_pump:=150;
                        ELSE
                                F_RAMP_pump:=1500; R_RAMP_pump:=TO_INT(PAR_NegFull_y);
                                IF  PWM_JOYY_L_UP>10 THEN
                                 F_RAMP_pump:=1500; R_RAMP_pump:=300;
                                END_IF
                        END_IF                
                4:
                        IF MainWinch_move AND (JiaYa_move OR CANO_JiayaPressure>80)  THEN
                                F_RAMP_pump:=1500; R_RAMP_pump:=150;
                        ELSE
                                F_RAMP_pump:=1500; R_RAMP_pump:=TO_INT(PAR_PosFull_y);//从200降
                                IF  PWM_JOYY_L_UP>10 THEN
                                 F_RAMP_pump:=1500; R_RAMP_pump:=300;
                                END_IF
                        END_IF                                
                5:
                        IF MainWinch_move AND (JiaYa_move OR CANO_JiayaPressure>80)  THEN
                                F_RAMP_pump:=1500; R_RAMP_pump:=200;
                        ELSE
                                F_RAMP_pump:=1500; R_RAMP_pump:=TO_INT(PAR_Zero_y);
                                IF  PWM_JOYY_L_UP>10 THEN
                                 F_RAMP_pump:=1500; R_RAMP_pump:=300;
                                END_IF
                        END_IF                        
                6:		IF MainWinch_move AND (JiaYa_move OR CANO_JiayaPressure>80)  THEN
                                F_RAMP_pump:=1500; R_RAMP_pump:=200;
                        ELSE
                                F_RAMP_pump:=1500; R_RAMP_pump:=200;
                                IF  PWM_JOYY_L_UP>10 THEN
                                 F_RAMP_pump:=1500; R_RAMP_pump:=300;
                                END_IF
                        END_IF  	
	END_CASE
(******斜坡增步长300 斜坡降步长300->400*****)	
RAMP15(
	IN:=UINT_TO_INT(RAMP15_IN), 
	ASCEND:= R_RAMP_pump, 
	DESCEND:= 1500, 
	TIMEBASE:=T#1000MS , 
	RESET:=FALSE , 
	OUT=>(PWM_Y1_SET));
(******减斜坡300->400*****)	
RAMP16(
	IN:=UINT_TO_INT(RAMP16_IN), 
	ASCEND:= R_RAMP_pump, 
	DESCEND:= 1500, 
	TIMEBASE:=T#1000MS , 
	RESET:=FALSE , 
	OUT=>(PWM_Y2_SET));


IF (NOT Rotation_move) AND (NOT MainWinch_move) AND (NOT PowerHead_move)
		AND (NOT JiaYa_move) AND (NOT ViceWinch_move)
		AND (NOT LeftMove_move) AND (NOT RightMove_move)  THEN
	PWM_Y1_Target:=0;
	PWM_Y2_Target:=0;
END_IF


IF PWM_Y1_SET<TO_INT(PAR_Y1_1_NegFull )THEN
	PWM_Y1_SET:=TO_INT(PAR_Y1_1_NegFull);
END_IF

IF PWM_Y2_SET<TO_INT(PAR_Y1_1_NegFull )THEN
	PWM_Y2_SET:=TO_INT(PAR_Y1_1_NegFull);
END_IF

IF(PWM_Y1_SET>1000) THEN
	PWM_Y1_SET := 300;
END_IF

IF(PWM_Y2_SET>1000) THEN
	PWM_Y2_SET := 300;
END_IF	

	PWM_Y8_SET_Target:=REAL_TO_UINT(UINT_TO_REAL(PWM_JOYY_L_UP)/1000*(PAR_Valve1_PosFull-PAR_Valve1_NegFull)+PAR_Valve1_NegFull);
	PWM_Y10_SET_Target:=REAL_TO_UINT(UINT_TO_REAL(PWM_JOYY_L_UP)/1000*(PAR_Valve2_PosFull-PAR_Valve2_NegFull)+PAR_Valve2_NegFull);
	PWM_Y7_SET_Target:=0;
	PWM_Y9_SET_Target:=0;
  //Y7 8 9 10处理	
		IF(PWM_Y8_SET<1000  AND  PWM_Y8_SET>=900)THEN    //主卷下放斜坡值
				F_RAMP_mainwinch_down:=200;
			
			ELSIF(PWM_Y8_SET<900)THEN
				F_RAMP_mainwinch_down:=400;
			ELSE
				F_RAMP_mainwinch_down:=400;
			END_IF
			
		IF(PWM_Y7_SET<1000  AND  PWM_Y7_SET>=900)THEN  //主卷上提斜坡值
				F_RAMP_mainwinch_down:=300;
		ELSIF(PWM_Y7_SET<900  )THEN
				F_RAMP_mainwinch_down:=200;
		ELSE
				F_RAMP_mainwinch_down:=400;
		END_IF
			
	RAMP7(
		IN:=WORD_TO_INT(PWM_Y7_SET_Target), 
		ASCEND:= R_RAMP_mainwinch, 
		DESCEND:= F_RAMP_mainwinch_up, 
		TIMEBASE:=TIMEBASE_mainwinch , 
		RESET:=FALSE , 
		OUT=>(PWM_Y7_SET_Target1));
	IF(PWM_Y7_SET_Target1>=400) THEN
		Curve_input:=TO_UINT(PWM_Y7_SET_Target1 - 400);
		IF(Curve_input>900) THEN
			Curve_input:=900;
		END_IF
		curve7(input:=REAL_TO_UINT(UINT_TO_REAL(Curve_input)*72.8),Zero:=FALSE,Full:=FALSE,
			   PAR_Progression:=Curve_Par,OutputEnable:=TRUE);
		PWM_Y7_SET:=PAR_Valve1_NegFull + REAL_TO_UINT(UINT_TO_REAL(curve7.Output)/72.8);
	ELSE
		PWM_Y7_SET:=0;
	END_IF
	
	
	RAMP8(
		IN:=WORD_TO_INT(PWM_Y8_SET_Target), 
		ASCEND:= R_RAMP_mainwinch, 
		DESCEND:= F_RAMP_mainwinch_down, 
		TIMEBASE:=TIMEBASE_mainwinch , 
		RESET:=FALSE , 
		OUT=>(PWM_Y8_SET_Target1));
	IF(PWM_Y8_SET_Target1>=400) THEN
		Curve_input:=TO_UINT(PWM_Y8_SET_Target1 - 400);
		IF(Curve_input>900) THEN
			Curve_input:=900;
		END_IF
		curve8(input:=REAL_TO_UINT(UINT_TO_REAL(Curve_input)*72.8),Zero:=FALSE,Full:=FALSE,
			   PAR_Progression:=Curve_Par,OutputEnable:=TRUE);
		PWM_Y8_SET:=PAR_Valve1_NegFull + REAL_TO_UINT(UINT_TO_REAL(curve8.Output)/72.8);
	ELSE
		PWM_Y8_SET:=0;
	END_IF
	
	
	RAMP9(
		IN:=WORD_TO_INT(PWM_Y9_SET_Target), 
		ASCEND:= R_RAMP_mainwinch, 
		DESCEND:= F_RAMP_mainwinch_up, 
		TIMEBASE:=TIMEBASE_mainwinch , 
		RESET:=FALSE , 
		OUT=>(PWM_Y9_SET_Target1));
	IF(PWM_Y9_SET_Target1>=400) THEN
		Curve_input:=TO_UINT(PWM_Y9_SET_Target1 - 400);
		IF(Curve_input>900) THEN
			Curve_input:=900;
		END_IF
		curve9(input:=REAL_TO_UINT(UINT_TO_REAL(Curve_input)*72.8),Zero:=FALSE,Full:=FALSE,
			   PAR_Progression:=Curve_Par,OutputEnable:=TRUE);
		PWM_Y9_SET:=PAR_Valve1_NegFull + REAL_TO_UINT(UINT_TO_REAL(curve9.Output)/72.8);
	ELSE
		PWM_Y9_SET:=0;
	END_IF
	
	RAMP10(
		IN:=WORD_TO_INT(PWM_Y10_SET_Target), 
		ASCEND:= R_RAMP_mainwinch, 
		DESCEND:= F_RAMP_mainwinch_down, 
		TIMEBASE:=TIMEBASE_mainwinch , 
		RESET:=FALSE , 
		OUT=>(PWM_Y10_SET_Target1));
	IF(PWM_Y10_SET_Target1>=400) THEN
		Curve_input:=TO_UINT(PWM_Y10_SET_Target1 - 400);
		IF(Curve_input>900) THEN
			Curve_input:=900;
		END_IF
		curve10(input:=REAL_TO_UINT(UINT_TO_REAL(Curve_input)*72.8),Zero:=FALSE,Full:=FALSE,
			   PAR_Progression:=Curve_Par,OutputEnable:=TRUE);
		PWM_Y10_SET:=PAR_Valve1_NegFull + REAL_TO_UINT(UINT_TO_REAL(curve10.Output)/72.8);
	ELSE
		PWM_Y10_SET:=0;
	END_IF
    //Y7 8 9 10范围限制
	IF(PWM_Y7_SET>1300)THEN
		PWM_Y7_SET :=1300;
	END_IF
	IF(PWM_Y8_SET>1300)THEN
		PWM_Y8_SET :=1300;
	END_IF
	IF(PWM_Y9_SET>1300)THEN
		PWM_Y9_SET :=1300;
	END_IF
	IF(PWM_Y10_SET>1300)THEN
		PWM_Y10_SET :=1300;
	END_IF
	
	IF(PWM_Y7_SET<=300)THEN
		PWM_Y7_SET :=0;
	END_IF
	IF(PWM_Y8_SET<=300)THEN
		PWM_Y8_SET :=0;
	END_IF
	IF(PWM_Y9_SET<=300)THEN
		PWM_Y9_SET :=0;
	END_IF
	IF(PWM_Y10_SET<=300)THEN
		PWM_Y10_SET :=0;
	END_IF
	
	PWM_Y7_SET:=0;
	PWM_Y9_SET:=0;
	(*主泵卸荷阀控制*)
		PWM_Y39_SET_Target:=MAX(PWM_Y8_SET_Target,PWM_Y7_SET_Target);
		PWM_Y40_SET_Target:=MAX(PWM_Y9_SET_Target,PWM_Y10_SET_Target);
	(*卸荷动作缓冲*)
RAMP19(
	IN:=WORD_TO_INT(PWM_Y39_SET_Target), 
	ASCEND:= R_RAMP_xiehe, 
	DESCEND:= F_RAMP_xiehe, 
	TIMEBASE:=TIMEBASE_xiehe , 
	RESET:=FALSE , 
	OUT=>(PWM_Y39_SET_Target1));
IF(PWM_Y39_SET_Target1>=400) THEN
	Curve_input:=TO_UINT(PWM_Y39_SET_Target1 - 400);
	IF(Curve_input>900) THEN
		Curve_input:=900;
	END_IF
	curve19(input:=REAL_TO_UINT(UINT_TO_REAL(Curve_input)*72.8),Zero:=FALSE,Full:=FALSE,
		   PAR_Progression:=Curve_Par1,OutputEnable:=TRUE);
	PWM_Y39_SET:=PAR_Valve1_NegFull + REAL_TO_UINT(UINT_TO_REAL(curve19.Output)/72.8);
ELSE
	PWM_Y39_SET:=0;
END_IF

RAMP20(
	IN:=WORD_TO_INT(PWM_Y40_SET_Target), 
	ASCEND:= R_RAMP_xiehe, 
	DESCEND:= F_RAMP_xiehe, 
	TIMEBASE:=TIMEBASE_xiehe , 
	RESET:=FALSE , 
	OUT=>(PWM_Y40_SET_Target1));
IF(PWM_Y40_SET_Target1>=400) THEN
	Curve_input:=TO_UINT(PWM_Y40_SET_Target1 - 400);
	IF(Curve_input>900) THEN
		Curve_input:=900;
	END_IF
	curve20(input:=REAL_TO_UINT(UINT_TO_REAL(Curve_input)*72.8),Zero:=FALSE,Full:=FALSE,
		   PAR_Progression:=Curve_Par1,OutputEnable:=TRUE);
	PWM_Y40_SET:=PAR_Valve1_NegFull + REAL_TO_UINT(UINT_TO_REAL(curve20.Output)/72.8);
ELSE
	PWM_Y40_SET:=0;
END_IF
	
IF(PWM_Y39_SET>1300)THEN
	PWM_Y39_SET :=1300;
END_IF
IF(PWM_Y40_SET>1300)THEN
	PWM_Y40_SET :=1300;
END_IF

IF(PWM_Y39_SET<=300)THEN
	PWM_Y39_SET :=0;
END_IF
IF(PWM_Y40_SET<=300)THEN
	PWM_Y40_SET :=0;
END_IF

END_PROGRAM

